
// ===== library: MasterCopy "Copy of Function blocks in 1. FB Bilbiotecas" =====

// folder: 1. FB Bilbiotecas

FUNCTION_BLOCK "FB BITS TO WORD"   // FB1, SCL
{ S7_Optimized_Access := 'TRUE' }
VERSION : 0.1
// Empacota 16 bools numa Word. Contrato consumido por gen-alarm-fc:
//  pinos de entrada SIGNAL_Bit0..SIGNAL_Bit15 e saida BITS_TO_WORD --
//  AlarmFc.RewireWordNetwork procura esses nomes exatos (AlarmFc.cs:313 e :348).
//  Renomear pino aqui quebra o gerador.
   VAR_INPUT
      SIGNAL_Bit0 : Bool;
      SIGNAL_Bit1 : Bool;
      SIGNAL_Bit2 : Bool;
      SIGNAL_Bit3 : Bool;
      SIGNAL_Bit4 : Bool;
      SIGNAL_Bit5 : Bool;
      SIGNAL_Bit6 : Bool;
      SIGNAL_Bit7 : Bool;
      SIGNAL_Bit8 : Bool;
      SIGNAL_Bit9 : Bool;
      SIGNAL_Bit10 : Bool;
      SIGNAL_Bit11 : Bool;
      SIGNAL_Bit12 : Bool;
      SIGNAL_Bit13 : Bool;
      SIGNAL_Bit14 : Bool;
      SIGNAL_Bit15 : Bool;
   END_VAR
   VAR_OUTPUT
      BITS_TO_WORD : Word;
   END_VAR
BEGIN

      // slice access: %X0 e o bit menos significativo da Word
      #BITS_TO_WORD.%X0 := #SIGNAL_Bit0;
      #BITS_TO_WORD.%X1 := #SIGNAL_Bit1;
      #BITS_TO_WORD.%X2 := #SIGNAL_Bit2;
      #BITS_TO_WORD.%X3 := #SIGNAL_Bit3;
      #BITS_TO_WORD.%X4 := #SIGNAL_Bit4;
      #BITS_TO_WORD.%X5 := #SIGNAL_Bit5;
      #BITS_TO_WORD.%X6 := #SIGNAL_Bit6;
      #BITS_TO_WORD.%X7 := #SIGNAL_Bit7;
      #BITS_TO_WORD.%X8 := #SIGNAL_Bit8;
      #BITS_TO_WORD.%X9 := #SIGNAL_Bit9;
      #BITS_TO_WORD.%X10 := #SIGNAL_Bit10;
      #BITS_TO_WORD.%X11 := #SIGNAL_Bit11;
      #BITS_TO_WORD.%X12 := #SIGNAL_Bit12;
      #BITS_TO_WORD.%X13 := #SIGNAL_Bit13;
      #BITS_TO_WORD.%X14 := #SIGNAL_Bit14;
      #BITS_TO_WORD.%X15 := #SIGNAL_Bit15;
END_FUNCTION_BLOCK

FUNCTION_BLOCK "FB BITS TO DOUBLE WORD"   // FB5, SCL
{ S7_Optimized_Access := 'TRUE' }
VERSION : 0.1
   VAR_INPUT
      SIGNAL_Bit0 : Bool;   // Sinal de entrada 1
      SIGNAL_Bit1 : Bool;   // Sinal de entrada 2
      SIGNAL_Bit2 : Bool;   // Sinal de entrada 3
      SIGNAL_Bit3 : Bool;   // Sinal de entrada 4
      SIGNAL_Bit4 : Bool;   // Sinal de entrada 5
      SIGNAL_Bit5 : Bool;   // Sinal de entrada 6
      SIGNAL_Bit6 : Bool;   // Sinal de entrada 7
      SIGNAL_Bit7 : Bool;   // Sinal de entrada 8
      SIGNAL_Bit8 : Bool;   // Sinal de entrada 9
      SIGNAL_Bit9 : Bool;   // Sinal de entrada 10
      SIGNAL_Bit10 : Bool;   // Sinal de entrada 11
      SIGNAL_Bit11 : Bool;   // Sinal de entrada 12
      SIGNAL_Bit12 : Bool;   // Sinal de entrada 13
      SIGNAL_Bit13 : Bool;   // Sinal de entrada 14
      SIGNAL_Bit14 : Bool;   // Sinal de entrada 15
      SIGNAL_Bit15 : Bool;   // Sinal de entrada 16
      SIGNAL_Bit16 : Bool;   // Sinal de entrada 17
      SIGNAL_Bit17 : Bool;   // Sinal de entrada 18
      SIGNAL_Bit18 : Bool;   // Sinal de entrada 19
      SIGNAL_Bit19 : Bool;   // Sinal de entrada 20
      SIGNAL_Bit20 : Bool;   // Sinal de entrada 21
      SIGNAL_Bit21 : Bool;   // Sinal de entrada 22
      SIGNAL_Bit22 : Bool;   // Sinal de entrada 23
      SIGNAL_Bit23 : Bool;   // Sinal de entrada 24
      SIGNAL_Bit24 : Bool;   // Sinal de entrada 25
      SIGNAL_Bit25 : Bool;   // Sinal de entrada 26
      SIGNAL_Bit26 : Bool;   // Sinal de entrada 27
      SIGNAL_Bit27 : Bool;   // Sinal de entrada 28
      SIGNAL_Bit28 : Bool;   // Sinal de entrada 29
      SIGNAL_Bit29 : Bool;   // Sinal de entrada 30
      SIGNAL_Bit30 : Bool;   // Sinal de entrada 31
      SIGNAL_Bit31 : Bool;   // Sinal de entrada 32
   END_VAR
   VAR_OUTPUT
      BITS_TO_DWORD : DWord;   // Word de saída com os sinais montados
   END_VAR
BEGIN
   // Word Alarmes - Montando bits em uma double word

   // Bits recebidos de campo
   #"BITS_TO_DWORD".%X0 := #SIGNAL_Bit0;
   #"BITS_TO_DWORD".%X1 := #SIGNAL_Bit1;
   #"BITS_TO_DWORD".%X2 := #SIGNAL_Bit2;
   #"BITS_TO_DWORD".%X3 := #SIGNAL_Bit3;
   #"BITS_TO_DWORD".%X4 := #SIGNAL_Bit4;
   #"BITS_TO_DWORD".%X5 := #SIGNAL_Bit5;
   #"BITS_TO_DWORD".%X6 := #SIGNAL_Bit6;
   #"BITS_TO_DWORD".%X7 := #SIGNAL_Bit7;
   #"BITS_TO_DWORD".%X8 := #SIGNAL_Bit8;
   #"BITS_TO_DWORD".%X9 := #SIGNAL_Bit9;
   #"BITS_TO_DWORD".%X10 := #SIGNAL_Bit10;
   #"BITS_TO_DWORD".%X11 := #SIGNAL_Bit11;
   #"BITS_TO_DWORD".%X12 := #SIGNAL_Bit12;
   #"BITS_TO_DWORD".%X13 := #SIGNAL_Bit13;
   #"BITS_TO_DWORD".%X14 := #SIGNAL_Bit14;
   #"BITS_TO_DWORD".%X15 := #SIGNAL_Bit15;
   #"BITS_TO_DWORD".%X16 := #SIGNAL_Bit16;
   #"BITS_TO_DWORD".%X17 := #SIGNAL_Bit17;
   #"BITS_TO_DWORD".%X18 := #SIGNAL_Bit18;
   #"BITS_TO_DWORD".%X19 := #SIGNAL_Bit19;
   #"BITS_TO_DWORD".%X20 := #SIGNAL_Bit20;
   #"BITS_TO_DWORD".%X21 := #SIGNAL_Bit21;
   #"BITS_TO_DWORD".%X22 := #SIGNAL_Bit22;
   #"BITS_TO_DWORD".%X23 := #SIGNAL_Bit23;
   #"BITS_TO_DWORD".%X24 := #SIGNAL_Bit24;
   #"BITS_TO_DWORD".%X25 := #SIGNAL_Bit25;
   #"BITS_TO_DWORD".%X26 := #SIGNAL_Bit26;
   #"BITS_TO_DWORD".%X27 := #SIGNAL_Bit27;
   #"BITS_TO_DWORD".%X28 := #SIGNAL_Bit28;
   #"BITS_TO_DWORD".%X29 := #SIGNAL_Bit29;
   #"BITS_TO_DWORD".%X30 := #SIGNAL_Bit30;
   #"BITS_TO_DWORD".%X31 := #SIGNAL_Bit31;
END_FUNCTION_BLOCK

FUNCTION_BLOCK "FB CONTADOR"   // FB7, LAD
TITLE = Function Block MINUTEIRO - Contador de Minutos
{ S7_Optimized_Access := 'TRUE' }
VERSION : 0.1
// Bloco para realizar a contagem de quantos minutos cada motor/bomba passou ligado.
   VAR_INPUT
      INPUT_LIGADO : Bool;   // Entrada do sinal de falha instanciado na Network 1
      INPUT_RESET_MINUTEIRO : Bool;   // Entrada do sinal de reset minuteiro (minutos trabalhadas da bomba)
   END_VAR
   VAR_OUTPUT
      SEGUNDEIRO : UInt;   // Saída do segundeiro (segundos trabalhados da bomba)
      MINUTEIRO : Real;   // Saída do minuteiro (minutos trabalhados da bomba)
      HORIMETRO : Real;   // Saída do horimetro (horas trabalhados da bomba)
   END_VAR
   VAR
      RESET_SEGUNDO : Bool;   // Comando para zerar os minutos acumuladas
      MINUTO : Bool;   // Pulso para contador de minutos
      COUNT_MINUTO : Bool;   // Contador de minutos
      RESET_MINUTO : Bool;   // Reset do contador de minutos
      SEGUNDOS : UInt;   // Segundos armazenados
      TIMER_SEGUNDO : IEC_COUNTER;   // Bloco contador de segundos
   END_VAR
BEGIN

REGION Network 1: Comando para zerar os minutos acumuladas
   // TIMER_SEGUNDO: Bloco contador de segundos
   // TIMER_MINUTO: Bloco contador de minutos
   // INC: Incremento de horas
   // RESET_MINUTEIRO: Comando para zerar os minutos acumulados
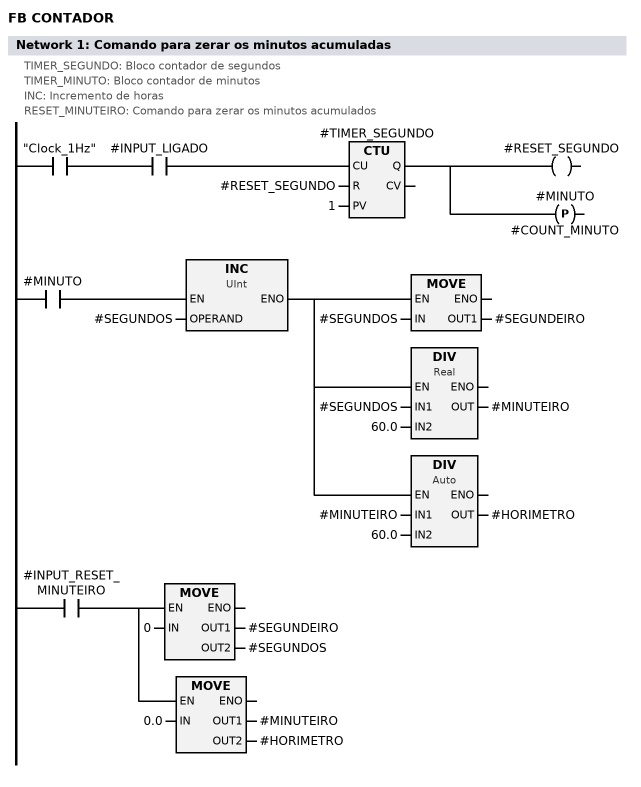
   #TIMER_SEGUNDO.CTU(CU := "Clock_1Hz" AND #INPUT_LIGADO, R := #RESET_SEGUNDO, PV := 1);
   #RESET_SEGUNDO := #TIMER_SEGUNDO.Q;
   #MINUTO := #TIMER_SEGUNDO.Q AND NOT #COUNT_MINUTO;   // rising edge
   #COUNT_MINUTO := #TIMER_SEGUNDO.Q;
   IF #MINUTO THEN
       #SEGUNDOS := #SEGUNDOS + 1;
       #SEGUNDEIRO := #SEGUNDOS;
       #MINUTEIRO := #SEGUNDOS / 60.0;
       #HORIMETRO := #MINUTEIRO / 60.0;
   END_IF;
   IF #INPUT_RESET_MINUTEIRO THEN
       #SEGUNDEIRO := 0;
       #SEGUNDOS := 0;
       #MINUTEIRO := 0.0;
       #HORIMETRO := 0.0;
   END_IF;
END_REGION
END_FUNCTION_BLOCK

FUNCTION_BLOCK "FB TOTALIZADOR"   // FB16, LAD
TITLE = Function Block TOTALIZADOR - Calculando os totalizadores dos macromedidores
{ S7_Optimized_Access := 'TRUE' }
VERSION : 0.1
// Network 1: Recebendo sinal de pulso
// Network 2: Primeira Soma (Incremento a cada 1 pulso)
// Network 3: Segunda Soma (Incremento a cada 1000 pulsos)
// Network 4: Resetando o totalizador
   VAR_INPUT
      ENTRADA_SINAL : Bool;   // Entrada do sinal proveniente do hidrômetro/macromedidor
      RESET_TOT : Bool;   // Input de reset para zerar os blocos de incremento do totalizador
      MULTIPLICADOR : Int;
   END_VAR
   VAR_OUTPUT
      TOT_SAÍDA : UInt;   // Saída real do totalizador (m³)
   END_VAR
   VAR RETAIN
      PULSE1 : Bool;   // Pulso inicial para contar os sinais elétricos da entrada digital
      COUNT_PULSE1 : Bool;   // Contador de Pulsos 1
      PULSE2 : Bool;   // Rampa de subida para assegurar que o sinal da comparação anterior seja identificado como pulso pelo CLP
      COUNT_PULSE2 : Bool;   // Contador de pulsos 2
      SOMA1 : UInt;   // Bloco de incremento a cada pulso recebido na variável PULSE
      SOMA1_TOT_PREV : UInt;   // Variável que recebe a primeira soma
      SOMA2 : UInt;   // Variável que recebe o incremento de 1000 em 1000 e move ao TOT_SAÍDA Output para ser utilizado
   END_VAR
   VAR
      MULT1 : UInt;
   END_VAR
BEGIN

REGION Network 1: Recebendo sinal de pulso
   // ENTRADA_SINAL: Input que recebe o sinal de pulso do equipamento
   // PULSE1: Rampa de subida para assegurar que o sinal recebido seja identificado como pulso pelo CLP
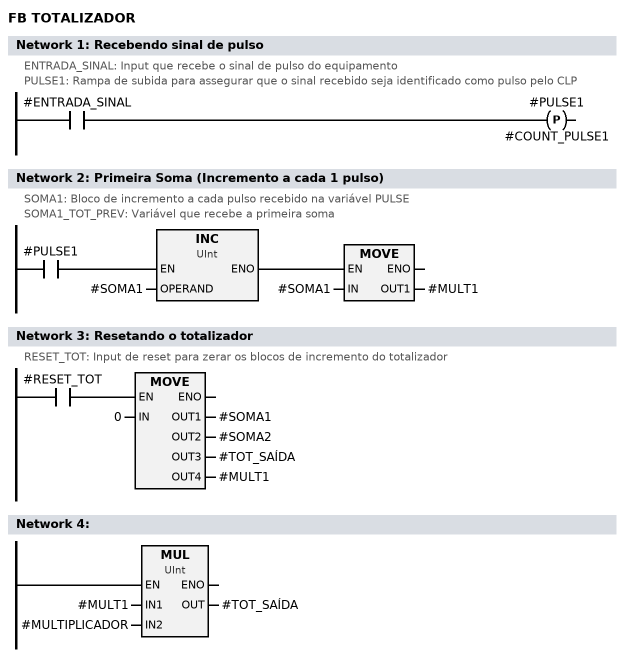
   #PULSE1 := #ENTRADA_SINAL AND NOT #COUNT_PULSE1;   // rising edge
   #COUNT_PULSE1 := #ENTRADA_SINAL;
END_REGION

REGION Network 2: Primeira Soma (Incremento a cada 1 pulso)
   // SOMA1: Bloco de incremento a cada pulso recebido na variável PULSE
   // SOMA1_TOT_PREV: Variável que recebe a primeira soma
   RUNG wire#powerrail
      Contact( #PULSE1 )
      { S7_Templates := "DestType := UInt" } Inc( #SOMA1 )
      Move(in := #SOMA1, out1 => #MULT1)
   END_RUNG
   // the same network as SCL:
   IF #PULSE1 THEN
       #SOMA1 := #SOMA1 + 1;
       #MULT1 := #SOMA1;
   END_IF;
END_REGION

REGION Network 3: Resetando o totalizador
   // RESET_TOT: Input de reset para zerar os blocos de incremento do totalizador
   RUNG wire#powerrail
      Contact( #RESET_TOT )
      Move(in := 0, out1 => #SOMA1, out2 => #SOMA2, out3 => #TOT_SAÍDA, out4 => #MULT1)
   END_RUNG
   // the same network as SCL:
   IF #RESET_TOT THEN
       #SOMA1 := 0;
       #SOMA2 := 0;
       #TOT_SAÍDA := 0;
       #MULT1 := 0;
   END_IF;
END_REGION

REGION Network 4
   RUNG wire#powerrail
      { S7_Templates := "SrcType := UInt" } Mul(in1 := #MULT1, in2 := #MULTIPLICADOR, out => #TOT_SAÍDA)
   END_RUNG
   // the same network as SCL:
   #TOT_SAÍDA := #MULT1 * #MULTIPLICADOR;
END_REGION
END_FUNCTION_BLOCK

FUNCTION_BLOCK "FB_HORÍMETRO"   // FB22, LAD
TITLE = Function Block HORÍMETRO - Contador de Horas
{ S7_Optimized_Access := 'TRUE' }
VERSION : 0.1
// Bloco para realizar a contagem de quantas horas cada motor/bomba passou ligado.
   VAR_INPUT
      INPUT_LIGADO : Bool;   // Entrada do sinal de falha instanciado na Network 1
      INPUT_RESET_HORIMETRO : Bool;   // Entrada do sinal de reset horímetro (horas trabalhadas da bomba)
   END_VAR
   VAR_OUTPUT
      HORIMETRO : UInt;   // Saída do horímetro (horas trabalhadas da bomba)
   END_VAR
   VAR RETAIN
      RESET_SEGUNDO : Bool;   // Comando para zerar as horas acumuladas
      MINUTO : Bool;   // Pulso para contador de minutos
      COUNT_MINUTO : Bool;   // Contador de minutos
      RESET_MINUTO : Bool;   // Reset do contador de minutos
      HORA : Bool;   // Pulso para contador de horas
      COUNT_HORA : Bool;   // Contador de horas
      HORAS : UInt;   // Horas armazenadas para mover ao Horimetro e zerar quando solicitado
      TIMER_SEGUNDO : IEC_COUNTER;   // Bloco contador de segundos
      TIMER_MINUTO : IEC_COUNTER;   // Bloco contador de minutos
   END_VAR
BEGIN

REGION Network 1: Acumulação de horas (Utilizando clock de 1Hz/1s)
   // TIMER_SEGUNDO: Bloco contador de segundos
   // TIMER_MINUTO: Bloco contador de minutos
   // INC: Incremento de horas
   // RESET_HORIMETRO: Comando para zerar as horas acumuladas
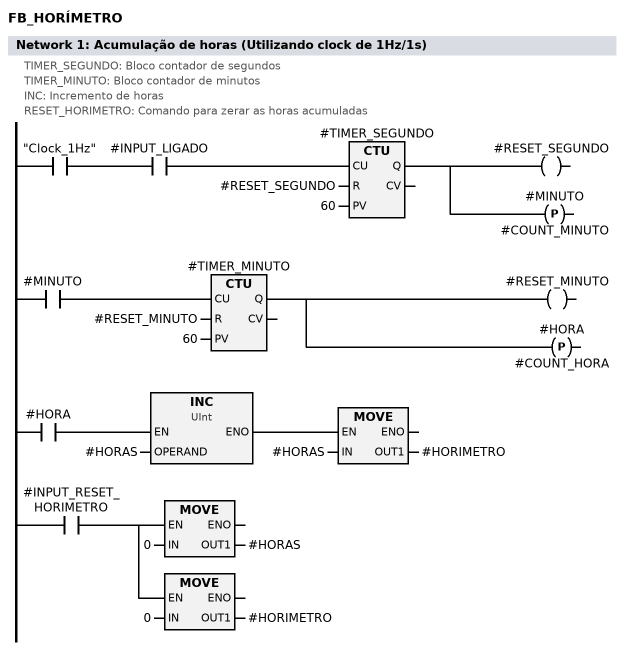
   #TIMER_SEGUNDO.CTU(CU := "Clock_1Hz" AND #INPUT_LIGADO, R := #RESET_SEGUNDO, PV := 60);
   #RESET_SEGUNDO := #TIMER_SEGUNDO.Q;
   #MINUTO := #TIMER_SEGUNDO.Q AND NOT #COUNT_MINUTO;   // rising edge
   #COUNT_MINUTO := #TIMER_SEGUNDO.Q;
   #TIMER_MINUTO.CTU(CU := #MINUTO, R := #RESET_MINUTO, PV := 60);
   #RESET_MINUTO := #TIMER_MINUTO.Q;
   #HORA := #TIMER_MINUTO.Q AND NOT #COUNT_HORA;   // rising edge
   #COUNT_HORA := #TIMER_MINUTO.Q;
   IF #HORA THEN
       #HORAS := #HORAS + 1;
       #HORIMETRO := #HORAS;
   END_IF;
   IF #INPUT_RESET_HORIMETRO THEN
       #HORAS := 0;
       #HORIMETRO := 0;
   END_IF;
END_REGION
END_FUNCTION_BLOCK

// folder: 1. FB Bilbiotecas/1.1 Acionamento

FUNCTION_BLOCK "FB CONDIÇÃO DE PARTIDA"   // FB6, LAD
TITLE = Function Block CONDIÇÃO DE PARTIDA - Intertravamentos para partir o motor/bomba
{ S7_Optimized_Access := 'TRUE' }
VERSION : 0.1
// Network 1: Gerenciamento Status Motor/Bomba
// Network 2: Recebimento dos sinais de entrada (Sinais de campo e comandos)
// Network 3: MODO MANUAL: Conjunto de condições para ligar e desligar
// Network 4: MODO AUTOMÁTICO: Conjunto de condições para ligar e desligar
// Network 5: FALHA: Condicionamento de falha
// Network 6: LIGA BOMBA: Validando intertravamentos para ligar
   VAR_INPUT
      INPUT_LIGADO : Bool;   // 1 = Sinal elétrico de campo indicando bomba ligada
      INPUT_DESLIGADO : Bool;   // 1 = Sinal elétrico de campo indicando bomba desligada
      INPUT_FALHA : Bool;   // 0 = Sinal elétrico de campo indicando bomba em falha
      INPUT_LOCAL_MAN : Bool;   // 1 = Sinal elétrico de campo indicando bomba em local
      INPUT_LOCAL_AUTO : Bool;   // 1 = Sinal elétrico de campo indicando bomba em local automático
      INPUT_REMOTO : Bool;   // 1 = Sinal elétrico de campo indicando bomba em remoto
      INPUT_FALHA_PROFINET : Bool;   // 1 = Indica falta de comunicação PROFINET com o equipamento
      INPUT_HABILITA_LIGA_AUTO : Bool;   // 1 = Sinal para habilitar Liga Bomba em Modo Automático quando todas as condições foram atentidas
      INPUT_CMD_LIGA : Bool;   // Comando enviado da IHM/SCADA para ligar a bomba
      CMD_MANUTEN : Bool;   // Comando enviado da IHM/SCADA para colocar a bomba em Modo de Manutenção
      CMD_MODO_OPERACAO : Bool;   // Comando enviado da IHM/SCADA para colocar a bomba em (0 = Modo Manual, 1 = Modo Automático)
      CMD_RESET_HORIMETRO : Bool;
   END_VAR
   VAR_OUTPUT
      LIGA_BOMBA : Bool;   // Saída acionada para ligar a bomba remotamente
      STATUS_MOTOR : Byte;   // 0 = DESLIGADO; 1 = LIGADO; 2 = FALHA; 3 = MANUTENÇÃO; 4 = SEM COMUNICAÇÃO MODBUS
      OUTPUT_REMOTO_AUTO : Bool;   // Saída para indicar bomba em Remoto Automático
      OUTPUT_MODO_OPER : Byte;
      STS_HORIMETRO : UInt;
      RESET_CMD_LIGA : Bool;
      STS_INTERTRAVAMENTO_AUTOMATICO : Bool;
   END_VAR
   VAR
      LOCAL_MAN : Bool;   // Saída para indicar bomba em Local Manual
      REMOTO_MAN : Bool;   // Saída para indicar bomba em Remoto Manual
      MANUTEN : Bool;   // Variável local para Indicar bomba em Modo Manutenção
      REMOTO : Bool;   // Variável local para indicar bomba em Modo Remoto
      FALHA : Bool;   // Variável local para indicar bomba em Falha
      LOCAL_AUTO : Bool;   // Variável local para indicar bomba em Modo Local Automático
      LIGA_REM_MAN : Bool;   // Variável local para Acionamento Remoto Manual
      LIGA_REM_AUTO : Bool;   // Variável local para Acionamento Remoto Automático
      "FB MODOS DE OPERAÇÃO_Instance" : "FB MODOS DE OPERAÇÃO";
      FB_HORÍMETRO_Instance : "FB_HORÍMETRO";
   END_VAR
   VAR_TEMP   // added for the SCL form of the ladder/FBD networks
      _w1 : Bool;
   END_VAR
BEGIN

REGION Network 1: Recebimento dos sinais de entrada (Sinais de campo e comandos)
   // INPUT_ABERTA = Entrada de sinal de Bomba Ligada
   // INPUT_FECHADA = Entrada de sinal de Bomba Desligada
   // INPUT_FALHA = Entrada de sinal de Bomba em Falha
   // INPUT_FALHA_PROFINET = Sem comunicação Profinet
   // STATUS_MOTOR: 0 = DESLIGADO; 1 = LIGADO; 2 = FALHA; 3 = MANUTENÇÃO; 4 = SEM COMUNICAÇÃO MODBUS
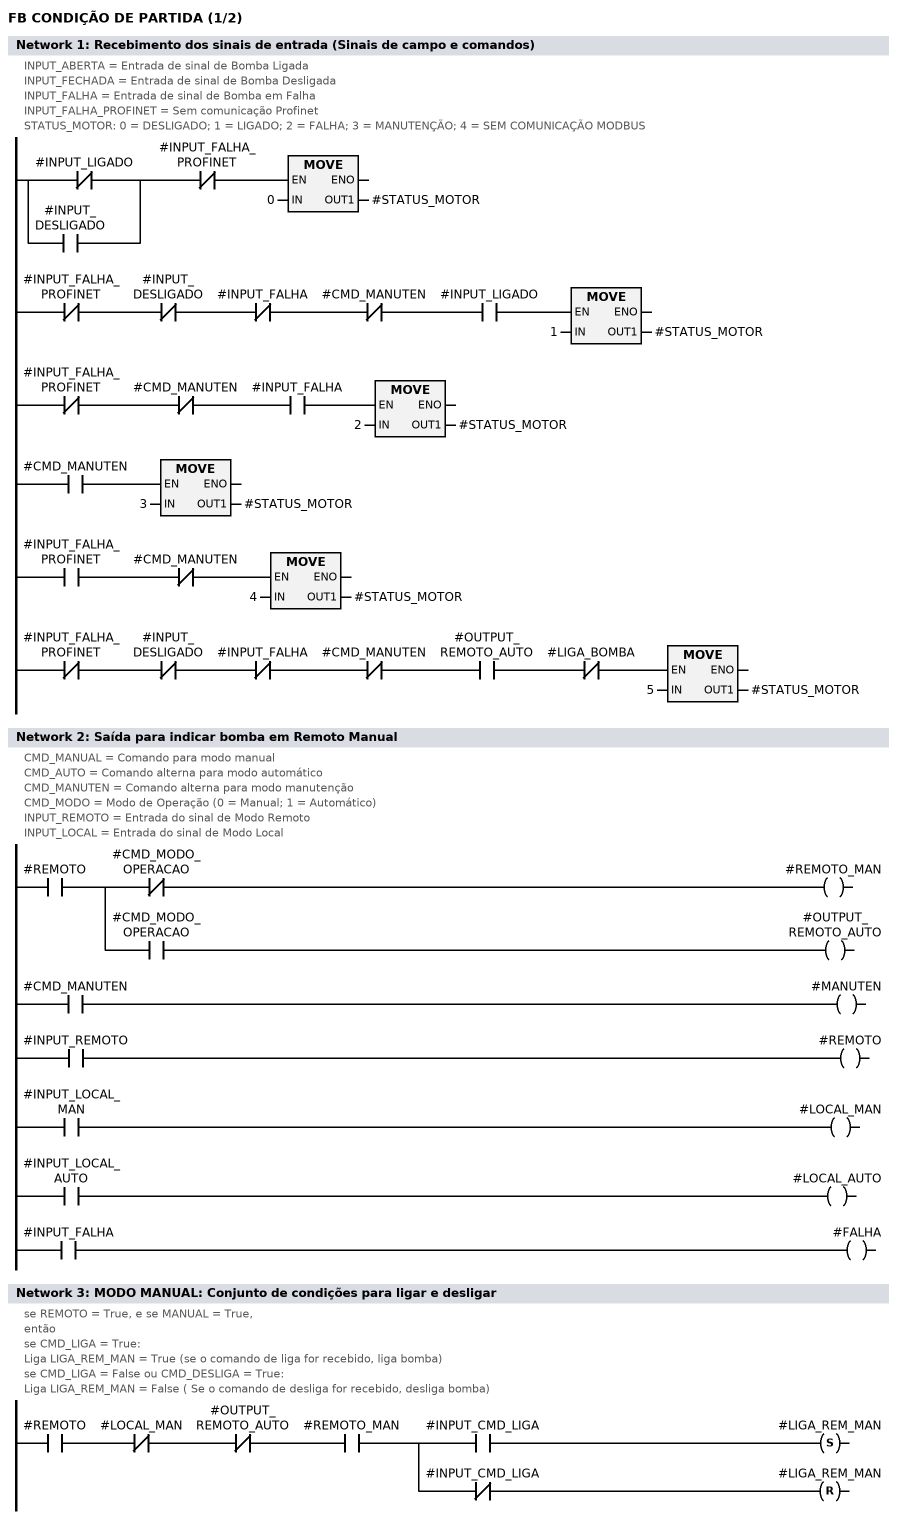
   RUNG wire#powerrail
      I_Contact( #INPUT_LIGADO )
      wire#w1
      I_Contact( #INPUT_FALHA_PROFINET )
      Move(in := 0, out1 => #STATUS_MOTOR)
   END_RUNG
   RUNG wire#powerrail
      Contact( #INPUT_DESLIGADO )
   END_RUNG wire#w1
   RUNG wire#powerrail
      I_Contact( #INPUT_FALHA_PROFINET )
      I_Contact( #INPUT_DESLIGADO )
      I_Contact( #INPUT_FALHA )
      I_Contact( #CMD_MANUTEN )
      Contact( #INPUT_LIGADO )
      Move(in := 1, out1 => #STATUS_MOTOR)
   END_RUNG
   RUNG wire#powerrail
      I_Contact( #INPUT_FALHA_PROFINET )
      I_Contact( #CMD_MANUTEN )
      Contact( #INPUT_FALHA )
      Move(in := 2, out1 => #STATUS_MOTOR)
   END_RUNG
   RUNG wire#powerrail
      Contact( #CMD_MANUTEN )
      Move(in := 3, out1 => #STATUS_MOTOR)
   END_RUNG
   RUNG wire#powerrail
      Contact( #INPUT_FALHA_PROFINET )
      I_Contact( #CMD_MANUTEN )
      Move(in := 4, out1 => #STATUS_MOTOR)
   END_RUNG
   RUNG wire#powerrail
      I_Contact( #INPUT_FALHA_PROFINET )
      I_Contact( #INPUT_DESLIGADO )
      I_Contact( #INPUT_FALHA )
      I_Contact( #CMD_MANUTEN )
      Contact( #OUTPUT_REMOTO_AUTO )
      I_Contact( #LIGA_BOMBA )
      Move(in := 5, out1 => #STATUS_MOTOR)
   END_RUNG
   // the same network as SCL:
   IF (NOT #INPUT_LIGADO OR #INPUT_DESLIGADO) AND NOT #INPUT_FALHA_PROFINET THEN #STATUS_MOTOR := 0; END_IF;
   IF NOT #INPUT_FALHA_PROFINET AND NOT #INPUT_DESLIGADO AND NOT #INPUT_FALHA AND NOT #CMD_MANUTEN AND #INPUT_LIGADO THEN
       #STATUS_MOTOR := 1;
   END_IF;
   IF NOT #INPUT_FALHA_PROFINET AND NOT #CMD_MANUTEN AND #INPUT_FALHA THEN #STATUS_MOTOR := 2; END_IF;
   IF #CMD_MANUTEN THEN #STATUS_MOTOR := 3; END_IF;
   IF #INPUT_FALHA_PROFINET AND NOT #CMD_MANUTEN THEN #STATUS_MOTOR := 4; END_IF;
   IF NOT #INPUT_FALHA_PROFINET AND NOT #INPUT_DESLIGADO AND NOT #INPUT_FALHA AND NOT #CMD_MANUTEN AND #OUTPUT_REMOTO_AUTO AND NOT #LIGA_BOMBA THEN
       #STATUS_MOTOR := 5;
   END_IF;
END_REGION

REGION Network 2: Saída para indicar bomba em Remoto Manual
   // CMD_MANUAL = Comando para modo manual
   // CMD_AUTO = Comando alterna para modo automático
   // CMD_MANUTEN = Comando alterna para modo manutenção
   // CMD_MODO = Modo de Operação (0 = Manual; 1 = Automático)
   // INPUT_REMOTO = Entrada do sinal de Modo Remoto
   // INPUT_LOCAL = Entrada do sinal de Modo Local
   RUNG wire#powerrail
      Contact( #REMOTO )
      wire#w1
      I_Contact( #CMD_MODO_OPERACAO )
      Coil( #REMOTO_MAN )
   END_RUNG
   RUNG wire#w1
      Contact( #CMD_MODO_OPERACAO )
      Coil( #OUTPUT_REMOTO_AUTO )
   END_RUNG
   RUNG wire#powerrail
      Contact( #CMD_MANUTEN )
      Coil( #MANUTEN )
   END_RUNG
   RUNG wire#powerrail
      Contact( #INPUT_REMOTO )
      Coil( #REMOTO )
   END_RUNG
   RUNG wire#powerrail
      Contact( #INPUT_LOCAL_MAN )
      Coil( #LOCAL_MAN )
   END_RUNG
   RUNG wire#powerrail
      Contact( #INPUT_LOCAL_AUTO )
      Coil( #LOCAL_AUTO )
   END_RUNG
   RUNG wire#powerrail
      Contact( #INPUT_FALHA )
      Coil( #FALHA )
   END_RUNG
   // the same network as SCL:
   #REMOTO_MAN := #REMOTO AND NOT #CMD_MODO_OPERACAO;
   #OUTPUT_REMOTO_AUTO := #REMOTO AND #CMD_MODO_OPERACAO;
   #MANUTEN := #CMD_MANUTEN;
   #REMOTO := #INPUT_REMOTO;
   #LOCAL_MAN := #INPUT_LOCAL_MAN;
   #LOCAL_AUTO := #INPUT_LOCAL_AUTO;
   #FALHA := #INPUT_FALHA;
END_REGION

REGION Network 3: MODO MANUAL: Conjunto de condições para ligar e desligar
   // se REMOTO = True, e se MANUAL = True,
   // 
   // então
   // se CMD_LIGA = True: 
   // Liga LIGA_REM_MAN = True (se o comando de liga for recebido, liga bomba)
   // 
   // se CMD_LIGA = False ou CMD_DESLIGA = True:
   // Liga LIGA_REM_MAN = False ( Se o comando de desliga for recebido, desliga bomba)
   RUNG wire#powerrail
      Contact( #REMOTO )
      I_Contact( #LOCAL_MAN )
      I_Contact( #OUTPUT_REMOTO_AUTO )
      Contact( #REMOTO_MAN )
      wire#w1
      Contact( #INPUT_CMD_LIGA )
      S_Coil( #LIGA_REM_MAN )
   END_RUNG
   RUNG wire#w1
      I_Contact( #INPUT_CMD_LIGA )
      R_Coil( #LIGA_REM_MAN )
   END_RUNG
   // the same network as SCL:
   #_w1 := #REMOTO AND NOT #LOCAL_MAN AND NOT #OUTPUT_REMOTO_AUTO AND #REMOTO_MAN;
   IF #_w1 AND #INPUT_CMD_LIGA THEN #LIGA_REM_MAN := TRUE; END_IF;
   IF #_w1 AND NOT #INPUT_CMD_LIGA THEN #LIGA_REM_MAN := FALSE; END_IF;
END_REGION

REGION Network 4: Variável local para Acionamento Remoto Auto
   // se REMOTO = True, e se AUTO = True:
   // 
   // então
   // se LIGA_REM_AUTO = True:
   // e se PARAMETRO < PARAMETRO_LIGA;
   // então LIGA_REM_AUTO = True (se a leitura for menor que o cadastro para ligar, liga em remoto automático)
   // 
   // se LIGA_REM_AUTO = False:
   // e se PARAMETRO >= PARAMETRO_DESLIGA:
   // então Desliga REMOTO AUTOMÁTICO (se a leitura for maior ou igual ao cadastro para desligar, desliga em remoto automático)
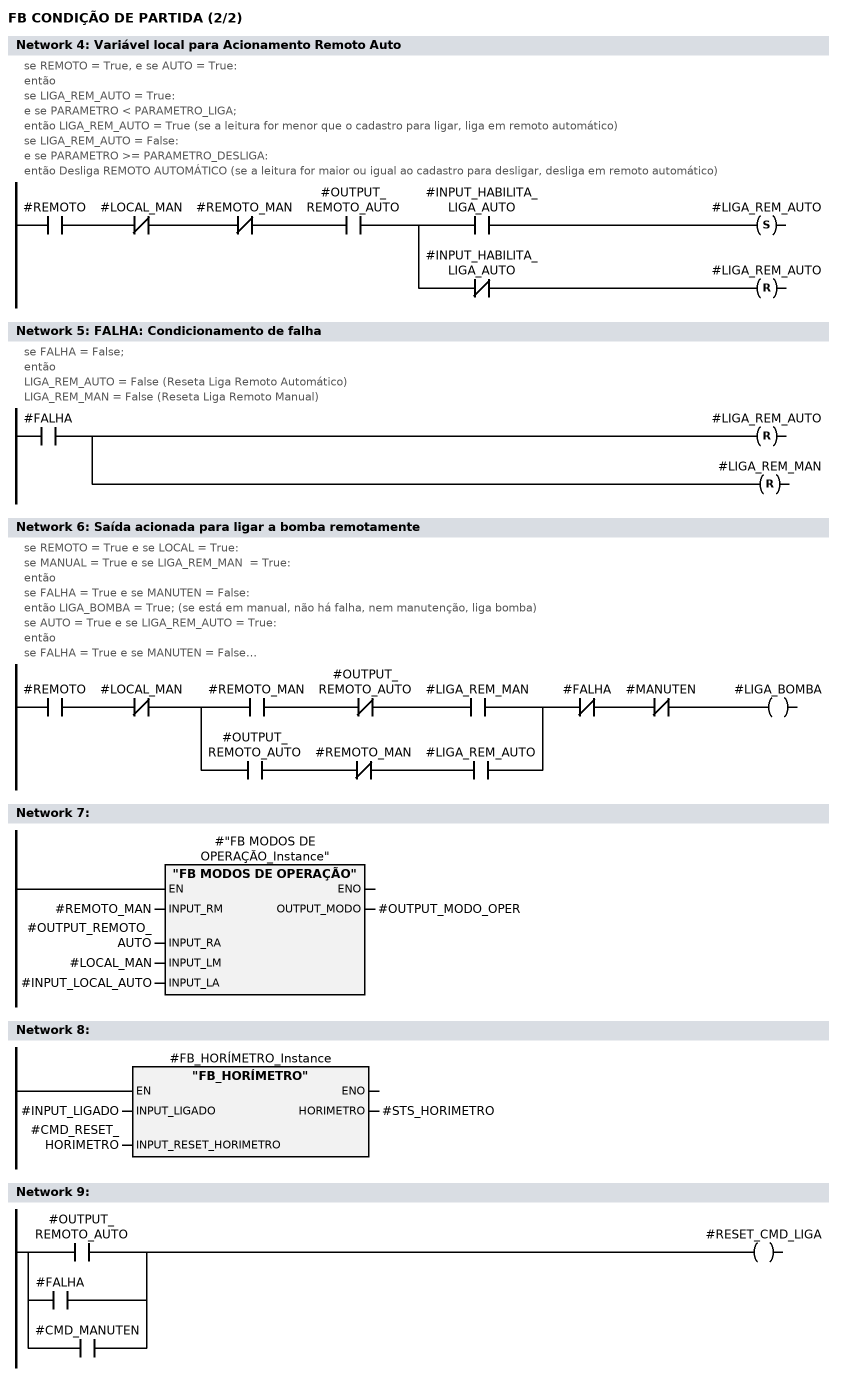
   RUNG wire#powerrail
      Contact( #REMOTO )
      I_Contact( #LOCAL_MAN )
      I_Contact( #REMOTO_MAN )
      Contact( #OUTPUT_REMOTO_AUTO )
      wire#w1
      Contact( #INPUT_HABILITA_LIGA_AUTO )
      S_Coil( #LIGA_REM_AUTO )
   END_RUNG
   RUNG wire#w1
      I_Contact( #INPUT_HABILITA_LIGA_AUTO )
      R_Coil( #LIGA_REM_AUTO )
   END_RUNG
   // the same network as SCL:
   #_w1 := #REMOTO AND NOT #LOCAL_MAN AND NOT #REMOTO_MAN AND #OUTPUT_REMOTO_AUTO;
   IF #_w1 AND #INPUT_HABILITA_LIGA_AUTO THEN #LIGA_REM_AUTO := TRUE; END_IF;
   IF #_w1 AND NOT #INPUT_HABILITA_LIGA_AUTO THEN #LIGA_REM_AUTO := FALSE; END_IF;
END_REGION

REGION Network 5: FALHA: Condicionamento de falha
   // se FALHA = False;
   // 
   // então
   // LIGA_REM_AUTO = False (Reseta Liga Remoto Automático)
   // LIGA_REM_MAN = False (Reseta Liga Remoto Manual)
   RUNG wire#powerrail
      Contact( #FALHA )
      wire#w1
      R_Coil( #LIGA_REM_AUTO )
   END_RUNG
   RUNG wire#w1
      R_Coil( #LIGA_REM_MAN )
   END_RUNG
   // the same network as SCL:
   IF #FALHA THEN
       #LIGA_REM_AUTO := FALSE;
       #LIGA_REM_MAN := FALSE;
   END_IF;
END_REGION

REGION Network 6: Saída acionada para ligar a bomba remotamente
   // se REMOTO = True e se LOCAL = True:
   // 
   // se MANUAL = True e se LIGA_REM_MAN  = True:
   // então
   // se FALHA = True e se MANUTEN = False:
   // então LIGA_BOMBA = True; (se está em manual, não há falha, nem manutenção, liga bomba)
   // 
   // se AUTO = True e se LIGA_REM_AUTO = True:
   // então
   // se FALHA = True e se MANUTEN = False:
   // então LIGA_BOMBA = True; (se está em automático, não há falha, nem manutenção, liga bomba)
   RUNG wire#powerrail
      Contact( #REMOTO )
      I_Contact( #LOCAL_MAN )
      wire#w1
      Contact( #REMOTO_MAN )
      I_Contact( #OUTPUT_REMOTO_AUTO )
      Contact( #LIGA_REM_MAN )
      wire#w2
      I_Contact( #FALHA )
      I_Contact( #MANUTEN )
      Coil( #LIGA_BOMBA )
   END_RUNG
   RUNG wire#w1
      Contact( #OUTPUT_REMOTO_AUTO )
      I_Contact( #REMOTO_MAN )
      Contact( #LIGA_REM_AUTO )
   END_RUNG wire#w2
   // the same network as SCL:
   #LIGA_BOMBA := #REMOTO AND NOT #LOCAL_MAN AND ((#REMOTO_MAN AND NOT #OUTPUT_REMOTO_AUTO AND #LIGA_REM_MAN) OR (#OUTPUT_REMOTO_AUTO AND NOT #REMOTO_MAN AND #LIGA_REM_AUTO)) AND NOT #FALHA AND NOT #MANUTEN;
END_REGION

REGION Network 7
   RUNG wire#powerrail
      #"FB MODOS DE OPERAÇÃO_Instance"(INPUT_RM := #REMOTO_MAN, INPUT_RA := #OUTPUT_REMOTO_AUTO, INPUT_LM := #LOCAL_MAN, INPUT_LA := #INPUT_LOCAL_AUTO, OUTPUT_MODO => #OUTPUT_MODO_OPER)
   END_RUNG
   // the same network as SCL:
   #"FB MODOS DE OPERAÇÃO_Instance"(INPUT_RM := #REMOTO_MAN,   // "FB MODOS DE OPERAÇÃO"
                           INPUT_RA := #OUTPUT_REMOTO_AUTO,
                           INPUT_LM := #LOCAL_MAN,
                           INPUT_LA := #INPUT_LOCAL_AUTO,
                           OUTPUT_MODO => #OUTPUT_MODO_OPER);
END_REGION

REGION Network 8
   RUNG wire#powerrail
      #FB_HORÍMETRO_Instance(INPUT_LIGADO := #INPUT_LIGADO, INPUT_RESET_HORIMETRO := #CMD_RESET_HORIMETRO, HORIMETRO => #STS_HORIMETRO)
   END_RUNG
   // the same network as SCL:
   #FB_HORÍMETRO_Instance(INPUT_LIGADO := #INPUT_LIGADO,   // "FB_HORÍMETRO"
                          INPUT_RESET_HORIMETRO := #CMD_RESET_HORIMETRO,
                          HORIMETRO => #STS_HORIMETRO);
END_REGION

REGION Network 9
   RUNG wire#powerrail
      Contact( #OUTPUT_REMOTO_AUTO )
      wire#w1
      Coil( #RESET_CMD_LIGA )
   END_RUNG
   RUNG wire#powerrail
      Contact( #FALHA )
   END_RUNG wire#w1
   RUNG wire#powerrail
      Contact( #CMD_MANUTEN )
   END_RUNG wire#w1
   // the same network as SCL:
   #RESET_CMD_LIGA := #OUTPUT_REMOTO_AUTO OR #FALHA OR #CMD_MANUTEN;
END_REGION
END_FUNCTION_BLOCK

FUNCTION_BLOCK "FB_LIGA/DESLIGA MODO AUTO"   // FB8, LAD
TITLE = Function Block LIGA/DESLIGA MODO AUTO
{ S7_Optimized_Access := 'TRUE' }
VERSION : 0.1
// Bloco para alternância dinâmica do tempo para ligar e desligar bomba.
// Network 1: Atribuição do sinal de liga
// Network 2: Function Block CONTADOR: Contador de tempo para bomba ligada
// Network 3: Comparativo de bomba ligada com tempo cadastrado para ficar ligada
// Network 4: Function Block CONTADOR: Contador de tempo para bomba desligada
// Network 5: Comparativo de bomba desligada com tempo cadastrado para ficar desligada
// Network 6: Transferindo sinal de bomba ligada/desligada para fora do bloco
   VAR_INPUT
      REMOTO_AUTO : Bool;   // Modo Remoto Automático
      CAD_TEMPO_LIGADA : Real;   // Cadastro tempo para bomba ficar ligada
      CAD_TEMPO_DESLIGADA : Real;   // Cadastro tempo para bomba ficar desligada
      TEMPO_ALTERNANCIA : Bool;   // Controle de alternancia entre bombas
   END_VAR
   VAR_OUTPUT
      HABILITA_LIGA_AUTO : Bool;   // Habilita Liga em Modo Automático
   END_VAR
   VAR_IN_OUT
      TEMPO_LIGADA_AUTO_SEG : Real;   // Tempo de bomba ligada em Modo Automático (segundos)
      TEMPO_LIGADA_AUTO_MIN : Real;   // Tempo de bomba ligada em Modo Automático (minutos)
      TEMPO_LIGADA_AUTO_HOR : Real;   // Tempo de bomba ligada em Modo Automático (horas)
      TEMPO_DESLIGADA_AUTO_SEG : Real;   // Tempo de bomba desligada em Modo Automático (segundos)
      TEMPO_DESLIGADA_AUTO_MIN : Real;   // Tempo de bomba desligada em Modo Automático (minutos)
      TEMPO_DESLIGADA_AUTO_HOR : Real;   // Tempo de bomba desligada em Modo Automático (horas)
   END_VAR
   VAR
      DESLIGA_AUTO : Bool;   // Desliga bomba em Modo Automático
      LIGA_AUTO : Bool;   // Liga bomba em Modo Automático
      MINUTEIRO_LIGADA : "FB CONTADOR";
      MINUTEIRO_DESLIGADA : "FB CONTADOR";
      TEMPO_LIGADA_AUTO_HORA : Bool;   // Tempo de bomba desligada em Modo Automático (em horas)
   END_VAR
BEGIN

REGION Network 1: Atribuição do sinal de liga
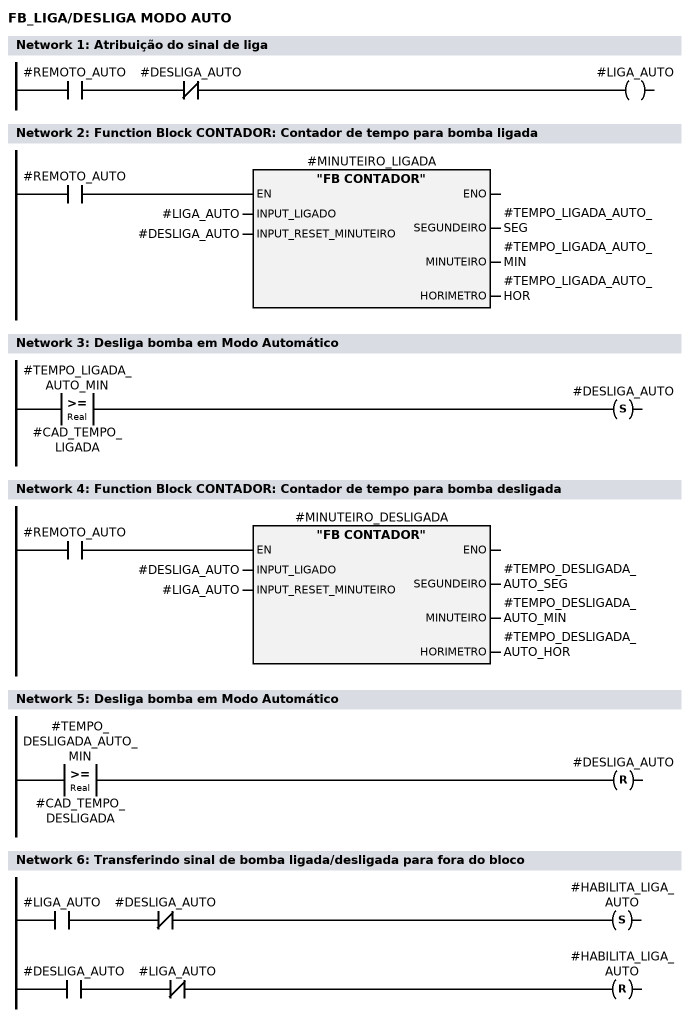
   RUNG wire#powerrail
      Contact( #REMOTO_AUTO )
      I_Contact( #DESLIGA_AUTO )
      Coil( #LIGA_AUTO )
   END_RUNG
   // the same network as SCL:
   #LIGA_AUTO := #REMOTO_AUTO AND NOT #DESLIGA_AUTO;
END_REGION

REGION Network 2: Function Block CONTADOR: Contador de tempo para bomba ligada
   RUNG wire#powerrail
      Contact( #REMOTO_AUTO )
      #MINUTEIRO_LIGADA(INPUT_LIGADO := #LIGA_AUTO, INPUT_RESET_MINUTEIRO := #DESLIGA_AUTO, SEGUNDEIRO => #TEMPO_LIGADA_AUTO_SEG, MINUTEIRO => #TEMPO_LIGADA_AUTO_MIN, HORIMETRO => #TEMPO_LIGADA_AUTO_HOR)
   END_RUNG
   // the same network as SCL:
   IF #REMOTO_AUTO THEN
       #MINUTEIRO_LIGADA(INPUT_LIGADO := #LIGA_AUTO,   // "FB CONTADOR"
                         INPUT_RESET_MINUTEIRO := #DESLIGA_AUTO,
                         SEGUNDEIRO => #TEMPO_LIGADA_AUTO_SEG,
                         MINUTEIRO => #TEMPO_LIGADA_AUTO_MIN,
                         HORIMETRO => #TEMPO_LIGADA_AUTO_HOR);
   END_IF;
END_REGION

REGION Network 3: Desliga bomba em Modo Automático
   RUNG wire#powerrail
      { S7_Templates := "SrcType := Real" } GE_Contact(in1 := #TEMPO_LIGADA_AUTO_MIN, in2 := #CAD_TEMPO_LIGADA)
      S_Coil( #DESLIGA_AUTO )
   END_RUNG
   // the same network as SCL:
   IF #TEMPO_LIGADA_AUTO_MIN >= #CAD_TEMPO_LIGADA THEN #DESLIGA_AUTO := TRUE; END_IF;
END_REGION

REGION Network 4: Function Block CONTADOR: Contador de tempo para bomba desligada
   RUNG wire#powerrail
      Contact( #REMOTO_AUTO )
      #MINUTEIRO_DESLIGADA(INPUT_LIGADO := #DESLIGA_AUTO, INPUT_RESET_MINUTEIRO := #LIGA_AUTO, SEGUNDEIRO => #TEMPO_DESLIGADA_AUTO_SEG, MINUTEIRO => #TEMPO_DESLIGADA_AUTO_MIN, HORIMETRO => #TEMPO_DESLIGADA_AUTO_HOR)
   END_RUNG
   // the same network as SCL:
   IF #REMOTO_AUTO THEN
       #MINUTEIRO_DESLIGADA(INPUT_LIGADO := #DESLIGA_AUTO,   // "FB CONTADOR"
                            INPUT_RESET_MINUTEIRO := #LIGA_AUTO,
                            SEGUNDEIRO => #TEMPO_DESLIGADA_AUTO_SEG,
                            MINUTEIRO => #TEMPO_DESLIGADA_AUTO_MIN,
                            HORIMETRO => #TEMPO_DESLIGADA_AUTO_HOR);
   END_IF;
END_REGION

REGION Network 5: Desliga bomba em Modo Automático
   RUNG wire#powerrail
      { S7_Templates := "SrcType := Real" } GE_Contact(in1 := #TEMPO_DESLIGADA_AUTO_MIN, in2 := #CAD_TEMPO_DESLIGADA)
      R_Coil( #DESLIGA_AUTO )
   END_RUNG
   // the same network as SCL:
   IF #TEMPO_DESLIGADA_AUTO_MIN >= #CAD_TEMPO_DESLIGADA THEN #DESLIGA_AUTO := FALSE; END_IF;
END_REGION

REGION Network 6: Transferindo sinal de bomba ligada/desligada para fora do bloco
   RUNG wire#powerrail
      Contact( #LIGA_AUTO )
      I_Contact( #DESLIGA_AUTO )
      S_Coil( #HABILITA_LIGA_AUTO )
   END_RUNG
   RUNG wire#powerrail
      Contact( #DESLIGA_AUTO )
      I_Contact( #LIGA_AUTO )
      R_Coil( #HABILITA_LIGA_AUTO )
   END_RUNG
   // the same network as SCL:
   IF #LIGA_AUTO AND NOT #DESLIGA_AUTO THEN #HABILITA_LIGA_AUTO := TRUE; END_IF;
   IF #DESLIGA_AUTO AND NOT #LIGA_AUTO THEN #HABILITA_LIGA_AUTO := FALSE; END_IF;
END_REGION
END_FUNCTION_BLOCK

FUNCTION_BLOCK "FB MODOS DE OPERAÇÃO"   // FB10, LAD
TITLE = Function Block MODOS DE OPERAÇÃO
{ S7_Optimized_Access := 'TRUE' }
VERSION : 0.1
// Movendo os valores booleados para uma variável do tipo int
   VAR_INPUT
      INPUT_RM : Bool;   // Entrada de sinal alto para indicar modo Remoto Manual
      INPUT_RA : Bool;   // Entrada de sinal alto para indicar modo Remoto Automático
      INPUT_LM : Bool;   // Entrada de sinal alto para indicar modo Local Manual
      INPUT_LA : Bool;   // Entrada de sinal alto para indicar modo Local Automático
   END_VAR
   VAR_OUTPUT
      OUTPUT_MODO : Int;   // Saída do Modo de Operação
   END_VAR
BEGIN

REGION Network 1: Estrutura de Operação
   // Se Remoto Manual = TRUE, OPERACAO_MOTOR = 1 
   // Se Remoto Automático = TRUE, OPERACAO_MOTOR = 2
   // Se Local Automático = TRUE, OPERACAO_MOTOR = 3
   // Se Local Manual = TRUE, OPERACAO_MOTOR = 4
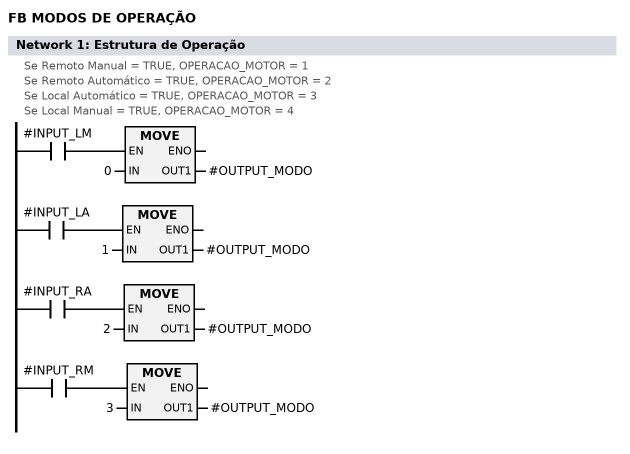
   RUNG wire#powerrail
      Contact( #INPUT_LM )
      Move(in := 0, out1 => #OUTPUT_MODO)
   END_RUNG
   RUNG wire#powerrail
      Contact( #INPUT_LA )
      Move(in := 1, out1 => #OUTPUT_MODO)
   END_RUNG
   RUNG wire#powerrail
      Contact( #INPUT_RA )
      Move(in := 2, out1 => #OUTPUT_MODO)
   END_RUNG
   RUNG wire#powerrail
      Contact( #INPUT_RM )
      Move(in := 3, out1 => #OUTPUT_MODO)
   END_RUNG
   // the same network as SCL:
   IF #INPUT_LM THEN #OUTPUT_MODO := 0; END_IF;
   IF #INPUT_LA THEN #OUTPUT_MODO := 1; END_IF;
   IF #INPUT_RA THEN #OUTPUT_MODO := 2; END_IF;
   IF #INPUT_RM THEN #OUTPUT_MODO := 3; END_IF;
END_REGION
END_FUNCTION_BLOCK

FUNCTION_BLOCK "FB_PARTIDA_INVERSOR"   // FB11, LAD
TITLE = Function Block PARTIDA INVERSOR
{ S7_Optimized_Access := 'TRUE' }
VERSION : 0.1
// Bloco para configurar os sinais de pulso (liga e desliga) em conjunto com 2 relés
   VAR_INPUT
      IN_LIGA_BOMBA : Bool;   // Entrada do comando para ligar a bomba
      IN_SUCÇÃO_OK : Bool;   // 0 = Sucção OK, permite ligar a bomba
      IN_OBSTRUÇÃO : Bool;   // 0 = Obstrução na pista
      IN_SOBRETORQUE : Bool;   // 0 = Sobretorque do motor/bomba
      IN_FALHA : Bool;   // 1 = Bomba em falha, comando desliga é pulsado
      IN_LIGADO : Bool;   // 1 = Bomba Ligada
      IN_HABILITA_CMB : Bool;   // Habilita bomba (Principal / Reserva)
      IN_LIGA_BOMBA_AUTO : Bool;
   END_VAR
   VAR_OUTPUT
      OUT_LIGA : Bool;   // Saída digital para ligar o Inversor
      OUT_DESLIGA : Bool;   // Saída digital para desligar o Inversor
   END_VAR
   VAR
      TEMP_LIGA : IEC_TIMER;   // Temporizador para simular o pulso de liga (0.5s)
      TEMP_DESLIGA : IEC_TIMER;   // Temporizador para simular o pulso de desliga (0.5s)
      DESLIGA_BOMBA : Bool;   // Memória auxiliar para desligar o Inversor
      OUT_TEST : Bool;
   END_VAR
BEGIN

REGION Network 1: Saída digital para ligar o Inversor
   // Condições para ligar:
   // IN_LIGA_BOMBA = 1, Sinal de liga recebido do bloco CONDIÇÃO DE PARTIDA
   // IN_SUCÇÃO = 1, Significa que a bomba está com sucção OK
   // IN_OBSTRUÇÃO = 0, Significa que não há obstrução na pista
   // IN_SOBRETORQUE = 0, Significa que não há alarme de sobretorque do motor/bomba
   // OUT_DESLIGA = 1, Para ligar, é necessário que a entrada digital de desliga no inversor (STOP) esteja com sinal alto, 
   // aguardando que o mesmo seja cortado com um pulso para desligar.
   // - Para desligar é necessário que o motor/bomba esteja enviando sinal de ligado.
   // 
   // Pulso para ligar: Configurado com um tempo de 0.5S
   // Pulso para desligar: Configurado com um tempo de 0.5S
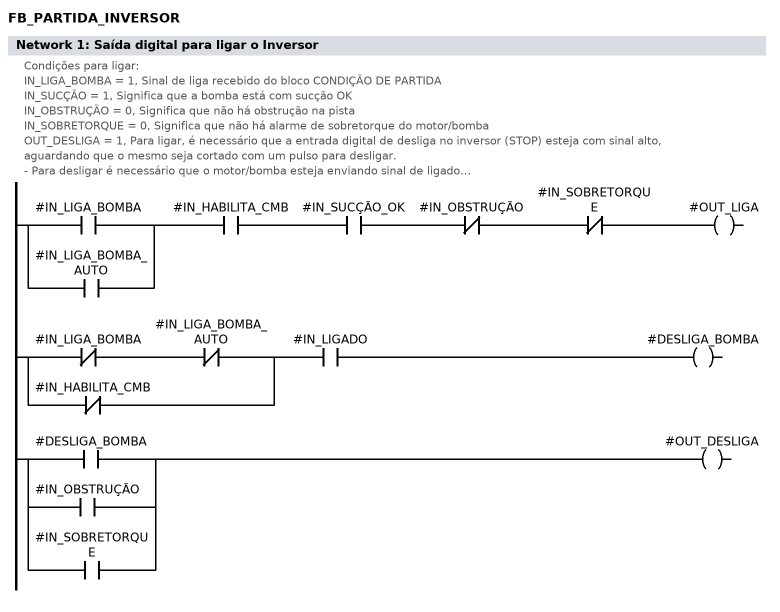
   RUNG wire#powerrail
      Contact( #IN_LIGA_BOMBA )
      wire#w1
      Contact( #IN_HABILITA_CMB )
      Contact( #IN_SUCÇÃO_OK )
      I_Contact( #IN_OBSTRUÇÃO )
      I_Contact( #IN_SOBRETORQUE )
      Coil( #OUT_LIGA )
   END_RUNG
   RUNG wire#powerrail
      Contact( #IN_LIGA_BOMBA_AUTO )
   END_RUNG wire#w1
   RUNG wire#powerrail
      I_Contact( #IN_LIGA_BOMBA )
      I_Contact( #IN_LIGA_BOMBA_AUTO )
      wire#w2
      Contact( #IN_LIGADO )
      Coil( #DESLIGA_BOMBA )
   END_RUNG
   RUNG wire#powerrail
      I_Contact( #IN_HABILITA_CMB )
   END_RUNG wire#w2
   RUNG wire#powerrail
      Contact( #DESLIGA_BOMBA )
      wire#w3
      Coil( #OUT_DESLIGA )
   END_RUNG
   RUNG wire#powerrail
      Contact( #IN_OBSTRUÇÃO )
   END_RUNG wire#w3
   RUNG wire#powerrail
      Contact( #IN_SOBRETORQUE )
   END_RUNG wire#w3
   // the same network as SCL:
   #OUT_LIGA := (#IN_LIGA_BOMBA OR #IN_LIGA_BOMBA_AUTO) AND #IN_HABILITA_CMB AND #IN_SUCÇÃO_OK AND NOT #IN_OBSTRUÇÃO AND NOT #IN_SOBRETORQUE;
   #DESLIGA_BOMBA := ((NOT #IN_LIGA_BOMBA AND NOT #IN_LIGA_BOMBA_AUTO) OR NOT #IN_HABILITA_CMB) AND #IN_LIGADO;
   #OUT_DESLIGA := #DESLIGA_BOMBA OR #IN_OBSTRUÇÃO OR #IN_SOBRETORQUE;
END_REGION
END_FUNCTION_BLOCK

FUNCTION_BLOCK "FB SUCÇÃO OK"   // FB15, LAD
TITLE = Function Block FB SUCÇÃO OK
{ S7_Optimized_Access := 'TRUE' }
VERSION : 0.1
   VAR_INPUT
      REFERENCIA : Real;   // Referência analógica em relação à sucção da bomba
      CADASTRO_SUCÇAO_INSUFICIENTE : Real;   // Cadastro de nível/pressão insuficiente
      CADASTRO_TEMPO_RESET : Time;   // Cadastro do tempo para resetar o alarme de Pressão Insuficiente
   END_VAR
   VAR_OUTPUT
      SUCÇÃO_OK : Bool;   // Sucção OK para operação
   END_VAR
   VAR
      SUCCAO_INSUFICIENTE : Bool;   // Sucção Insuficiente para operação
      RESET_ALARME : IEC_TIMER;   // Reset alarme de Sucção Insuficiente
   END_VAR
BEGIN

REGION Network 1: Set e Reset da Referência de Sucção insuficiente
   // Se nível for menor que a referência do Reservatório SUCÇÃO INSUFICIENTE,  bomba não pode ligar.
   // Caso o Nivel seja maior que a refêrencia então, após tempo cadastrado a bomba está habita para ligar
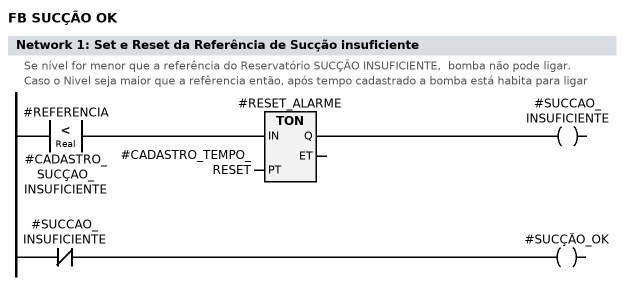
   #RESET_ALARME.TON(IN := #REFERENCIA < #CADASTRO_SUCÇAO_INSUFICIENTE, PT := #CADASTRO_TEMPO_RESET);
   #SUCCAO_INSUFICIENTE := #RESET_ALARME.Q;
   #SUCÇÃO_OK := NOT #SUCCAO_INSUFICIENTE;
END_REGION
END_FUNCTION_BLOCK

FUNCTION_BLOCK "FB VALVULA"   // FB17, LAD
{ S7_Optimized_Access := 'TRUE' }
VERSION : 0.1
// Network 1: Gerenciamento Status Válvula
// Network 2: Recebimento dos sinais de entrada (Sinais de campo e comandos)
// Network 3: MODO MANUAL: Conjunto de condições para ligar e desligar
// Network 4: MODO AUTOMÁTICO: Conjunto de condições para ligar e desligar
// Network 5: FALHA: Condicionamento de falha
// Network 6: LIGA BOMBA: Validando intertravamentos para ligar
// Network 7: ABRE VÁLVULA: Validando intertravamentos para abrir
   VAR_INPUT
      INPUT_ABERTA : Bool;   // 1 = Sinal elétrico de campo indicando válvula aberta
      INPUT_FECHADA : Bool;   // 1 = Sinal elétrico de campo indicando válvula fechada
      INPUT_FALHA : Bool;   // 0 = Sinal elétrico de campo indicando válvula em falha
      INPUT_LOCAL : Bool;   // 1 = Sinal elétrico de campo indicando válvula em modo local
      INPUT_REMOTO : Bool;   // 1 = Sinal elétrico de campo indicando válvula em modo remoto
      INPUT_FALHA_PROFINET : Bool;   // 1 = Indica falta de comunicação PROFINET com o equipamento
      INPUT_LIGA_AUTO : Bool;   // 1= indica que o processo pode ser ligado remoto manual
      PARAMETRO_ABRE : Bool;   // Parâmetro utilizado para abrir a válvula em modo automático
      PARAMETRO_FECHA : Bool;   // Parâmetro utilizado para fechar a válvula em modo automático
      CMD_ABRE : Bool;   // Comando enviado da IHM/SCADA para abrir a válvula
      CMD_MANUTEN : Bool;   // Comando enviado da IHM/SCADA para colocar a válvula em Modo de Manutenção
      CMD_MODO : Bool;   // Comando enviado da IHM/SCADA para colocar a bomba em (0 = Modo Manual, 1 = Modo Automático)
   END_VAR
   VAR_OUTPUT
      STATUS_VALV : Byte;   // 0 = FECHADA; 1 = ABERTA; 2 = FALHA
      ABRE_VALVULA : Bool;   // Saída acionada para abrir a válvula remotamente
      FECHA_VALVULA : Bool;   // Saída acionada para fechar a válvula remotamente
      REMOTO_MAN : Bool;   // Modo de Operação Remoto Manual
      REMOTO_AUTO : Bool;   // Modo de Operação Remoto Automático
      LOCAL_MAN : Bool;   // Modo de Operação Local Manual
   END_VAR
   VAR
      MANUTEN : Bool;   // Variável local para Indicar bomba em Modo Manutenção
      REMOTO : Bool;   // Variável local para indicar Modo Remoto
      FALHA : Bool;   // Variável local para Válvula em Falha
      ABRE_REM_MAN : Bool;   // Variável local para Acionamento Remoto Manual
      ABRE_REM_AUTO : Bool;   // Variável local para Acionamento Remoto Automático
   END_VAR
   VAR_TEMP   // added for the SCL form of the ladder/FBD networks
      _w1 : Bool;
   END_VAR
BEGIN

REGION Network 1: Gerenciamento Status Válvula
   // INPUT_ABERTA = Entrada de sinal de Válvula Aberta
   // INPUT_FECHADA = Entrada de sinal de Válvula Fechada
   // INPUT_FALHA = Entrada de sinal de Válvula em Falha
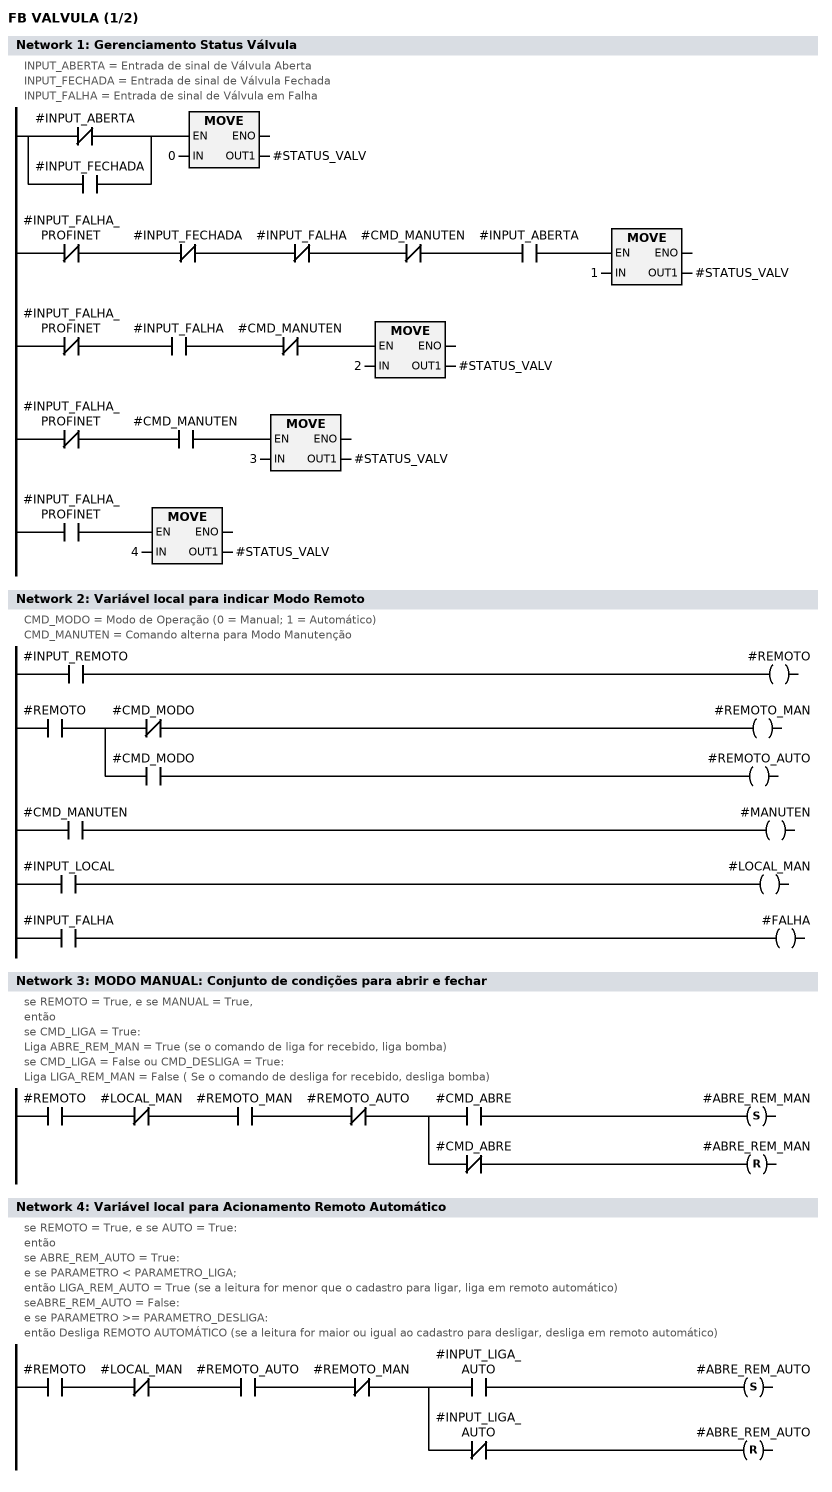
   RUNG wire#powerrail
      I_Contact( #INPUT_ABERTA )
      wire#w1
      Move(in := 0, out1 => #STATUS_VALV)
   END_RUNG
   RUNG wire#powerrail
      Contact( #INPUT_FECHADA )
   END_RUNG wire#w1
   RUNG wire#powerrail
      I_Contact( #INPUT_FALHA_PROFINET )
      I_Contact( #INPUT_FECHADA )
      I_Contact( #INPUT_FALHA )
      I_Contact( #CMD_MANUTEN )
      Contact( #INPUT_ABERTA )
      Move(in := 1, out1 => #STATUS_VALV)
   END_RUNG
   RUNG wire#powerrail
      I_Contact( #INPUT_FALHA_PROFINET )
      Contact( #INPUT_FALHA )
      I_Contact( #CMD_MANUTEN )
      Move(in := 2, out1 => #STATUS_VALV)
   END_RUNG
   RUNG wire#powerrail
      I_Contact( #INPUT_FALHA_PROFINET )
      Contact( #CMD_MANUTEN )
      Move(in := 3, out1 => #STATUS_VALV)
   END_RUNG
   RUNG wire#powerrail
      Contact( #INPUT_FALHA_PROFINET )
      Move(in := 4, out1 => #STATUS_VALV)
   END_RUNG
   // the same network as SCL:
   IF NOT #INPUT_ABERTA OR #INPUT_FECHADA THEN #STATUS_VALV := 0; END_IF;
   IF NOT #INPUT_FALHA_PROFINET AND NOT #INPUT_FECHADA AND NOT #INPUT_FALHA AND NOT #CMD_MANUTEN AND #INPUT_ABERTA THEN
       #STATUS_VALV := 1;
   END_IF;
   IF NOT #INPUT_FALHA_PROFINET AND #INPUT_FALHA AND NOT #CMD_MANUTEN THEN #STATUS_VALV := 2; END_IF;
   IF NOT #INPUT_FALHA_PROFINET AND #CMD_MANUTEN THEN #STATUS_VALV := 3; END_IF;
   IF #INPUT_FALHA_PROFINET THEN #STATUS_VALV := 4; END_IF;
END_REGION

REGION Network 2: Variável local para indicar Modo Remoto
   // CMD_MODO = Modo de Operação (0 = Manual; 1 = Automático)
   // CMD_MANUTEN = Comando alterna para Modo Manutenção
   RUNG wire#powerrail
      Contact( #INPUT_REMOTO )
      Coil( #REMOTO )
   END_RUNG
   RUNG wire#powerrail
      Contact( #REMOTO )
      wire#w1
      I_Contact( #CMD_MODO )
      Coil( #REMOTO_MAN )
   END_RUNG
   RUNG wire#w1
      Contact( #CMD_MODO )
      Coil( #REMOTO_AUTO )
   END_RUNG
   RUNG wire#powerrail
      Contact( #CMD_MANUTEN )
      Coil( #MANUTEN )
   END_RUNG
   RUNG wire#powerrail
      Contact( #INPUT_LOCAL )
      Coil( #LOCAL_MAN )
   END_RUNG
   RUNG wire#powerrail
      Contact( #INPUT_FALHA )
      Coil( #FALHA )
   END_RUNG
   // the same network as SCL:
   #REMOTO := #INPUT_REMOTO;
   #REMOTO_MAN := #REMOTO AND NOT #CMD_MODO;
   #REMOTO_AUTO := #REMOTO AND #CMD_MODO;
   #MANUTEN := #CMD_MANUTEN;
   #LOCAL_MAN := #INPUT_LOCAL;
   #FALHA := #INPUT_FALHA;
END_REGION

REGION Network 3: MODO MANUAL: Conjunto de condições para abrir e fechar
   // se REMOTO = True, e se MANUAL = True,
   // 
   // então
   // se CMD_LIGA = True: 
   // Liga ABRE_REM_MAN = True (se o comando de liga for recebido, liga bomba)
   // 
   // se CMD_LIGA = False ou CMD_DESLIGA = True:
   // Liga LIGA_REM_MAN = False ( Se o comando de desliga for recebido, desliga bomba)
   RUNG wire#powerrail
      Contact( #REMOTO )
      I_Contact( #LOCAL_MAN )
      Contact( #REMOTO_MAN )
      I_Contact( #REMOTO_AUTO )
      wire#w1
      Contact( #CMD_ABRE )
      S_Coil( #ABRE_REM_MAN )
   END_RUNG
   RUNG wire#w1
      I_Contact( #CMD_ABRE )
      R_Coil( #ABRE_REM_MAN )
   END_RUNG
   // the same network as SCL:
   #_w1 := #REMOTO AND NOT #LOCAL_MAN AND #REMOTO_MAN AND NOT #REMOTO_AUTO;
   IF #_w1 AND #CMD_ABRE THEN #ABRE_REM_MAN := TRUE; END_IF;
   IF #_w1 AND NOT #CMD_ABRE THEN #ABRE_REM_MAN := FALSE; END_IF;
END_REGION

REGION Network 4: Variável local para Acionamento Remoto Automático
   // se REMOTO = True, e se AUTO = True:
   // 
   // então
   // se ABRE_REM_AUTO = True:
   // e se PARAMETRO < PARAMETRO_LIGA;
   // então LIGA_REM_AUTO = True (se a leitura for menor que o cadastro para ligar, liga em remoto automático)
   // 
   // seABRE_REM_AUTO = False:
   // e se PARAMETRO >= PARAMETRO_DESLIGA:
   // então Desliga REMOTO AUTOMÁTICO (se a leitura for maior ou igual ao cadastro para desligar, desliga em remoto automático)
   RUNG wire#powerrail
      Contact( #REMOTO )
      I_Contact( #LOCAL_MAN )
      Contact( #REMOTO_AUTO )
      I_Contact( #REMOTO_MAN )
      wire#w1
      Contact( #INPUT_LIGA_AUTO )
      S_Coil( #ABRE_REM_AUTO )
   END_RUNG
   RUNG wire#w1
      I_Contact( #INPUT_LIGA_AUTO )
      R_Coil( #ABRE_REM_AUTO )
   END_RUNG
   // the same network as SCL:
   #_w1 := #REMOTO AND NOT #LOCAL_MAN AND #REMOTO_AUTO AND NOT #REMOTO_MAN;
   IF #_w1 AND #INPUT_LIGA_AUTO THEN #ABRE_REM_AUTO := TRUE; END_IF;
   IF #_w1 AND NOT #INPUT_LIGA_AUTO THEN #ABRE_REM_AUTO := FALSE; END_IF;
END_REGION

REGION Network 5: FALHA: Condicionamento de falha
   // se FALHA = False;
   // 
   // então
   // ABRE_REM_AUTO = False (Reseta Liga Remoto Automático)
   // ABRE_REM_MAN = False (Reseta Liga Remoto Manual)
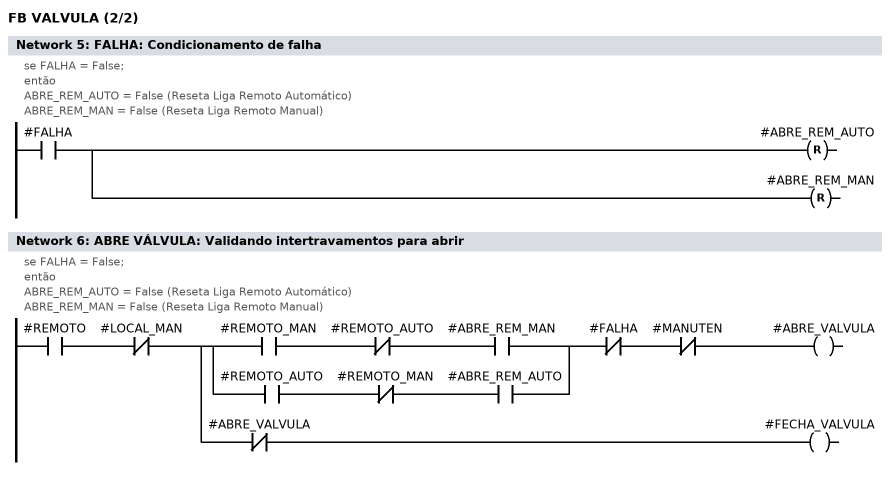
   RUNG wire#powerrail
      Contact( #FALHA )
      wire#w1
      R_Coil( #ABRE_REM_AUTO )
   END_RUNG
   RUNG wire#w1
      R_Coil( #ABRE_REM_MAN )
   END_RUNG
   // the same network as SCL:
   IF #FALHA THEN
       #ABRE_REM_AUTO := FALSE;
       #ABRE_REM_MAN := FALSE;
   END_IF;
END_REGION

REGION Network 6: ABRE VÁLVULA: Validando intertravamentos para abrir
   // se FALHA = False;
   // 
   // então
   // ABRE_REM_AUTO = False (Reseta Liga Remoto Automático)
   // ABRE_REM_MAN = False (Reseta Liga Remoto Manual)
   RUNG wire#powerrail
      Contact( #REMOTO )
      I_Contact( #LOCAL_MAN )
      wire#w1
      Contact( #REMOTO_MAN )
      I_Contact( #REMOTO_AUTO )
      Contact( #ABRE_REM_MAN )
      wire#w2
      I_Contact( #FALHA )
      I_Contact( #MANUTEN )
      Coil( #ABRE_VALVULA )
   END_RUNG
   RUNG wire#w1
      Contact( #REMOTO_AUTO )
      I_Contact( #REMOTO_MAN )
      Contact( #ABRE_REM_AUTO )
   END_RUNG wire#w2
   RUNG wire#w1
      I_Contact( #ABRE_VALVULA )
      Coil( #FECHA_VALVULA )
   END_RUNG
   // the same network as SCL:
   #_w1 := #REMOTO AND NOT #LOCAL_MAN;
   #ABRE_VALVULA := #_w1 AND ((#REMOTO_MAN AND NOT #REMOTO_AUTO AND #ABRE_REM_MAN) OR (#REMOTO_AUTO AND NOT #REMOTO_MAN AND #ABRE_REM_AUTO)) AND NOT #FALHA AND NOT #MANUTEN;
   #FECHA_VALVULA := #_w1 AND NOT #ABRE_VALVULA;
END_REGION
END_FUNCTION_BLOCK

FUNCTION_BLOCK "FB INTERTRAVAMENTO_PAINEL"   // FB27, SCL
{ S7_Optimized_Access := 'TRUE' }
VERSION : 0.1
   VAR_INPUT
      INPUT_BT_EMERGENCIA : Bool;
      INPUT_DISJUNTOR : Bool;
      INPUT_FONTE1 : Bool;
      INPUT_FONTE2 : Bool;
      INPUT_RELE_FALTA : Bool;
      INPUT_CONDICAO : Bool;
      INPUT_TESTE : Bool;
   END_VAR
   VAR_OUTPUT
      OUTPUT_PAINEL_OK : Bool;
   END_VAR
BEGIN

   IF ((#INPUT_BT_EMERGENCIA AND // Supondo que BT_EMERGENCIA é True quando ñ ATUADO
         NOT #INPUT_DISJUNTOR AND
         #INPUT_FONTE1 AND
         #INPUT_FONTE2 AND
         #INPUT_RELE_FALTA AND // Supondo que RELE_FALTA é True quando ñ ATUADO
         #INPUT_CONDICAO) 
      OR
      #INPUT_TESTE) THEN // teste força a saída 
   #OUTPUT_PAINEL_OK := TRUE;
   ELSE
       #OUTPUT_PAINEL_OK := FALSE;
   END_IF;
END_FUNCTION_BLOCK

// folder: 1. FB Bilbiotecas/1.1 Acionamento/1.1.1 Inversores

FUNCTION_BLOCK "FB AFERIÇÃO INVERSORES"   // FB2, LAD
{ S7_Optimized_Access := 'TRUE' }
VERSION : 0.1
// Os sinais de campo são recebidos em corrente (4-20mA) e representados pelo fundo de escala do CLP. Este bloco faz a conversão do sinal para a leitura real da medição.
// 
// Network 1: Ajuste do fundo de escala aos parâmetros de aferição
// Network 2: Cálculo da equação da reta para definir a leitura atual da entrada analógica
// Network 3: Setando o alarme SEM 4mA na entrada digital caso seja rompida
   VAR_INPUT
      ANALOG_IN_4a20mA : Int;   // Entrada do sinal analógico
      Y1_CONFIG : Int;   // Fundo de escala mínimo para o CLP
      Y2_CONFIG : Int;   // Fundo de escala máximo para o CLP
      X1_CONFIG : Int;   // Fundo de escala mínimo para o equipamento
      X2_CONFIG : Int;   // Fundo de escala máximo para o equipamento
      COMANDO : Int;   // Comando enviado da IHM/SCADA para aferir determinado equipamento
      COMANDO_VALOR : Int;   // Valor comparativo para executar o Bloco FB
      GRANDEZA_MAX : Int;   // Referência a grandeza maxima no qual o bloco vai utilizar para fazer a curva da reta
   END_VAR
   VAR_OUTPUT
      ANALOG_OUT_4a20mA : Real;   // Saída do sinal analógico já aferido
      ALARME_SEM_4mA : Bool;   // 1 = Entrada sem 4mA, indicando erro; 0 = Entrada OK
      RANGE_MIN_CADASTRADO : Int;   // Valor do cadastro máximo armazenado para visualizar na IHM
      RANGE_MAX_CADASTRADO : Int;   // Valor do cadastro mínimo armazenado para visualizar na IHM
   END_VAR
   VAR
      ANALOG_IN_LIMITED : Int;   // Tratamento de erro do sinal analógico para capturar apenas leituras que estão dentro do range do CLP
      ANALOG_IN_LIMITED_REAL : UInt;   // Saída do sinal ajustado conforme a grandeza máxima
      STATIC_X1 : UInt;   // Fundo de escala mínimo para o equipamento (Instanciado no FB)
      STATIC_X2 : UInt;   // Fundo de escala máximo para o equipamento (Instanciado no FB)
      STATIC_Y1 : UInt;   // Fundo de escala mínimo para o CLP (Instanciado no FB)
      STATIC_Y2 : UInt;   // Fundo de escala máximo para o CLP (Instanciado no FB)
      STATIC_GRANDEZA_MAX : UInt;   // Grandeza máxima do equipamento
      AJUSTAR_CURVA : Bool;   // Memória para mover as entradas às instâncias
      PONTO_ZERO : Int;   // Range mínimo do equipamento quando é diferente de 0
      ALARME_RESET : TOF_TIME;   // Reset do alarme Sem 4mA ao estabilizar o sinal
      PULSO_AJUSTAR : Bool;   // Pulso para realizar a aferição da curva
   END_VAR
   VAR_TEMP   // added for the SCL form of the ladder/FBD networks
      _w1 : Bool;
   END_VAR
BEGIN

REGION Network 1: Ajuste do fundo de escala aos parâmetros de aferição
   // X1_CONFIG = Fundo de escala mínimo para o equipamento
   // X2_CONFIG = Fundo de escala máximo para o equipamento
   // Y1_CONFIG = Fundo de escala mínimo para o CLP
   // Y2_CONFIG = Fundo de escala máximo para o CLP
   // GRANDEZA_MAX = Referência a grandeza maxima no qual o bloco vai utilizar para fazer a curva da reta
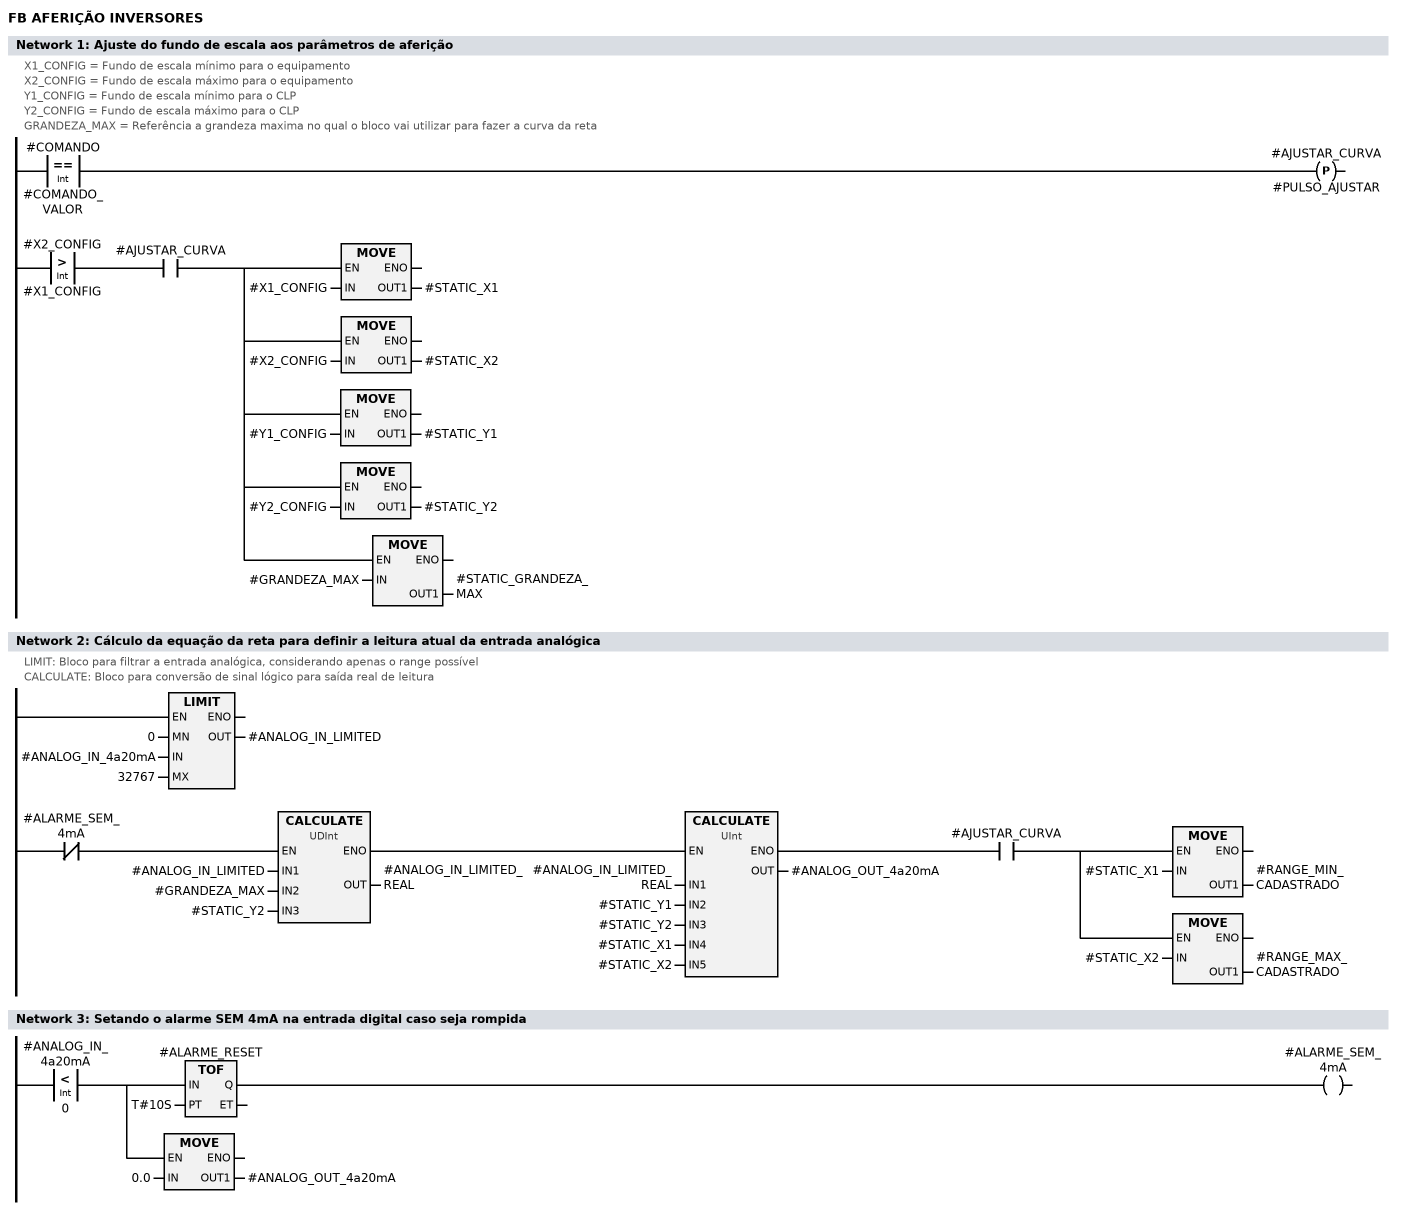
   #_w1 := #COMANDO = #COMANDO_VALOR;
   #AJUSTAR_CURVA := #_w1 AND NOT #PULSO_AJUSTAR;   // rising edge
   #PULSO_AJUSTAR := #_w1;
   IF (#X2_CONFIG > #X1_CONFIG) AND #AJUSTAR_CURVA THEN
       #STATIC_X1 := #X1_CONFIG;
       #STATIC_X2 := #X2_CONFIG;
       #STATIC_Y1 := #Y1_CONFIG;
       #STATIC_Y2 := #Y2_CONFIG;
       #STATIC_GRANDEZA_MAX := #GRANDEZA_MAX;
   END_IF;
END_REGION

REGION Network 2: Cálculo da equação da reta para definir a leitura atual da entrada analógica
   // LIMIT: Bloco para filtrar a entrada analógica, considerando apenas o range possível
   // CALCULATE: Bloco para conversão de sinal lógico para saída real de leitura
   #ANALOG_IN_LIMITED := LIMIT(MN := 0, IN := #ANALOG_IN_4a20mA, MX := 32767);
   IF NOT #ALARME_SEM_4mA THEN
       #ANALOG_IN_LIMITED_REAL := #ANALOG_IN_LIMITED * #STATIC_Y2 / #GRANDEZA_MAX;
       #ANALOG_OUT_4a20mA := (#ANALOG_IN_LIMITED_REAL - #STATIC_Y1) * (#STATIC_X2 - #STATIC_X1) / (#STATIC_Y2 - #STATIC_Y1);
   END_IF;
   IF NOT #ALARME_SEM_4mA AND #AJUSTAR_CURVA THEN
       #RANGE_MIN_CADASTRADO := #STATIC_X1;
       #RANGE_MAX_CADASTRADO := #STATIC_X2;
   END_IF;
END_REGION

REGION Network 3: Setando o alarme SEM 4mA na entrada digital caso seja rompida
   #_w1 := #ANALOG_IN_4a20mA < 0;
   #ALARME_RESET(IN := #_w1, PT := T#10S);   // TOF
   #ALARME_SEM_4mA := #ALARME_RESET.Q;
   IF #_w1 THEN #ANALOG_OUT_4a20mA := 0.0; END_IF;
END_REGION
END_FUNCTION_BLOCK

FUNCTION_BLOCK "FB STATUS ECSX"   // FB12, LAD
TITLE = Function Block STATUS ECSX - Status dos exaustores (ECS1 - ECS2 - ECS3)
{ S7_Optimized_Access := 'TRUE' }
VERSION : 0.1
// Sinais de status (ligado e falha) recebidos de campo
   VAR_INPUT
      INPUT_LIGADO : Bool;   // Entrada do sinal de Motor/Bomba ligado
      INPUT_FALHA : Bool;   // Entrada do sinal de falha instanciado na Network 1
      INPUT_MANUTEN : Bool;   // Entrada do sinal de manutenção instanciado na Network 1
      INPUT_FALHA_PROFINET : Bool;   // 1 = Indica falta de comunicação PROFINET com o equipamento
   END_VAR
   VAR_OUTPUT
      STATUS_MOTOR : Byte;   // Indicador de Status do exaustor
   END_VAR
BEGIN

REGION Network 1: Acionamento do status ligado
   // INUPT_LIGADO = TRUE: Exaustor ligado
   // INPUT_FALHA = TRUE: Exaustor em falha
   // INPUT_FALHA_PROFINET = TRUE: Sem Comunicação PROFINET
   // INPUT_MANUTEN = TRUE: Motor/Exaustor em manutenção
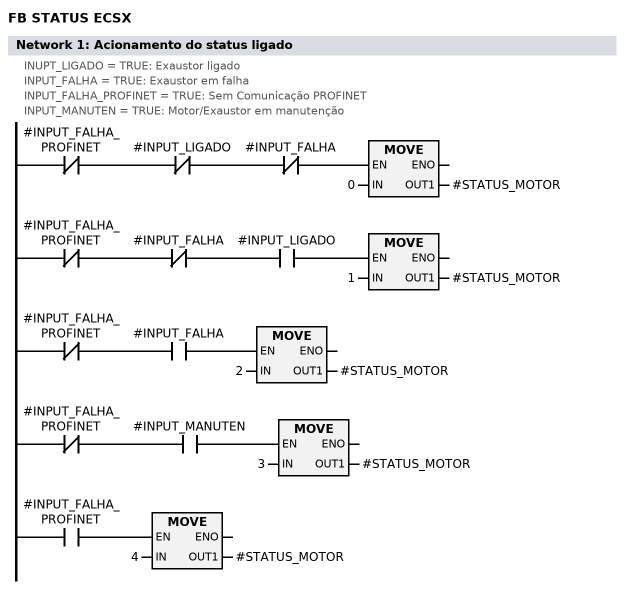
   RUNG wire#powerrail
      I_Contact( #INPUT_FALHA_PROFINET )
      I_Contact( #INPUT_LIGADO )
      I_Contact( #INPUT_FALHA )
      Move(in := 0, out1 => #STATUS_MOTOR)
   END_RUNG
   RUNG wire#powerrail
      I_Contact( #INPUT_FALHA_PROFINET )
      I_Contact( #INPUT_FALHA )
      Contact( #INPUT_LIGADO )
      Move(in := 1, out1 => #STATUS_MOTOR)
   END_RUNG
   RUNG wire#powerrail
      I_Contact( #INPUT_FALHA_PROFINET )
      Contact( #INPUT_FALHA )
      Move(in := 2, out1 => #STATUS_MOTOR)
   END_RUNG
   RUNG wire#powerrail
      I_Contact( #INPUT_FALHA_PROFINET )
      Contact( #INPUT_MANUTEN )
      Move(in := 3, out1 => #STATUS_MOTOR)
   END_RUNG
   RUNG wire#powerrail
      Contact( #INPUT_FALHA_PROFINET )
      Move(in := 4, out1 => #STATUS_MOTOR)
   END_RUNG
   // the same network as SCL:
   IF NOT #INPUT_FALHA_PROFINET AND NOT #INPUT_LIGADO AND NOT #INPUT_FALHA THEN #STATUS_MOTOR := 0; END_IF;
   IF NOT #INPUT_FALHA_PROFINET AND NOT #INPUT_FALHA AND #INPUT_LIGADO THEN #STATUS_MOTOR := 1; END_IF;
   IF NOT #INPUT_FALHA_PROFINET AND #INPUT_FALHA THEN #STATUS_MOTOR := 2; END_IF;
   IF NOT #INPUT_FALHA_PROFINET AND #INPUT_MANUTEN THEN #STATUS_MOTOR := 3; END_IF;
   IF #INPUT_FALHA_PROFINET THEN #STATUS_MOTOR := 4; END_IF;
END_REGION
END_FUNCTION_BLOCK

FUNCTION_BLOCK "FB INVERSOR SIEMENS"   // FB20, LAD
{ S7_Optimized_Access := 'TRUE' }
VERSION : 0.1
   VAR_INPUT
      RPM_min_Driver : Int;
      RPM_Max_Driver : Int;
      Setpoint_Velocidade : Int;
   END_VAR
   VAR_OUTPUT
      Telegram_Out_Velocidade : Int;
   END_VAR
   VAR_TEMP
      Aux_Velocidade : Real;
   END_VAR
BEGIN

REGION Network 1: Controle Velocidade
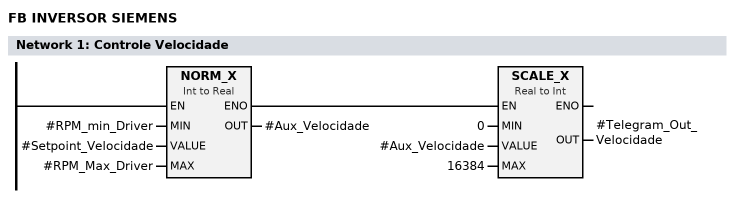
   RUNG wire#powerrail
      { S7_Templates := "[SrcType := Int, DestType := Real]" } Normalize(min := #RPM_min_Driver, value := #Setpoint_Velocidade, max := #RPM_Max_Driver, out => #Aux_Velocidade)
      { S7_Templates := "[SrcType := Real, DestType := Int]" } Scale(min := 0, value := #Aux_Velocidade, max := 16384, out => #Telegram_Out_Velocidade)
   END_RUNG
   // the same network as SCL:
   #Aux_Velocidade := NORM_X(MIN := #RPM_min_Driver, VALUE := #Setpoint_Velocidade, MAX := #RPM_Max_Driver);
   #Telegram_Out_Velocidade := SCALE_X(MIN := 0, VALUE := #Aux_Velocidade, MAX := 16384);
END_REGION
END_FUNCTION_BLOCK

FUNCTION_BLOCK "SINA_SPEED_TLG20"   // FB38003, SCL
TITLE = Speed control S7 to SINAMICS using Standardtelegram 20
{ S7_Optimized_Access := 'TRUE' }
AUTHOR : SIEMENS
FAMILY : DRIVES
NAME : SINA_SPD_TLG20
VERSION : 1.0
// The function block SINA_SPEED_TLG20 controls a SINAMICS drive using standard telegram 20
   VAR_INPUT
      enableAxis : Bool;   // 0 -> 1 = Enable the drive (OFF2 / OFF 3 are 1 in default status) (OFF1 = 0->1)
      ackError : Bool;   // 0 -> 1 = Acknowledge drive error
      speedSp : Real;   // Speed setpoint [rpm]
      selectCDS : USInt;   // Selection of the Command Data Set (0 = CDS0, 1 = CDS1)
      refSpeed : Real;   // Reference speed [p2000] in [rpm]
      refCurrent : Real;   // Reference current [p2002] in [Aeff]
      refTorque : Real;   // Reference torque [p2003] in [Nm]
      refPower : Real;   // Reference power [r2005] in [kW]
      configAxis : Word := 16#003F;   // binary programmed input to control all functions in the telegram without its own function block input
      HWIDSTW : HW_IO;   // Hardware Identifer set point slot
      HWIDZSW : HW_IO;   // Hardware Identifer actual value slot
   END_VAR
   VAR_OUTPUT
      axisEnabled : Bool;   // 1 = Drive is enabled
      lockout : Bool;   // 1 = Drive lockout active
      actCDS : USInt;   // Active Command Data Set (0 = CDS0, 1 = CDS1)
      actSpeed : Real;   // Smoothed actual speed in [1/min]
      actCurrent : Real;   // Smoothed current actual in [Arms]
      actTorque : Real;   // Actual smoothed torque in [Nm]
      actPower : Real;   // Actual smoothed active power in [kW]
      faultVIKNAMUR : Word;   // Fault word according to the VIK-NAMUR defintion
      error : Bool;   // 1 = Error (FB and Infeed)
      status : Int;   // Status output (7002 = FB in operation; 7xxx = warning; 8xxx = error description - read the manual)
      diagId : Int;   // Error codes of the system function blocks DPWR / DPRD_DAT
   END_VAR
   VAR_TEMP
      tempSpeed : Real;   // Speed setpoint in percent
      tempRefValueInvalid : Bool;   // At least one reference value is 0 or < 0
      tempSendBuf : Array[0..1] of Word;   // Send buffer
      tempRecvBuf : Array[0..5] of Word;   // Receive buffer
   END_VAR
   VAR CONSTANT
      NORMALIZATION_VALUE : Int := 16#4000;   // Used to calculate the Real values
      MAX_INT : Int := 16#7FFF;
      MIN_INT : Int := 16#8000;
      REF_CURRRENT_INVALID : Int := 16#7010;   // RefCurrent input is 0 or < 0
      REF_TORQUE_INVALID : Int := 16#7011;   // RefTorque input is 0 or < 0
      REF_POWER_INVALID : Int := 16#7012;   // RefPower input is 0 or < 0
      REF_VALUES_INVALID : Int := 16#7013;   // Multiple reference values are 0 or < 0
      NO_ERROR : Int := 16#7002;   // No error
      ERROR_REF_SPEED_INVALID : Int := 16#8001;   // RefSpeed input is 0 or < 0
      ERROR_INVALID_CDS : Int := 16#8002;   // Invalid Command Data Set selected
      ERROR_DRIVE : Int := 16#8401;   // Drive error
      ERROR_LOCKOUT : Int := 16#8402;   // Drive lockout
      ERROR_DPREAD : Int := 16#8600;   // DPRD_DAT returned an error
      ERROR_DPWRITE : Int := 16#8601;   // DPWR_DAT returned an error
      ERROR_FAULT_WORD : Int := 16#8700;   // faultVIKNAMUR is not 0
      STW1 : USInt := 0;
      ZSW1 : USInt := 0;
      NSOLL_A : USInt := 1;
   END_VAR
BEGIN
   //=============================================================================
   //SIEMENS AG
   //(c)Copyright 2019 All Rights Reserved
   //-----------------------------------------------------------------------------
   // Library:       LSINAExt
   // Tested with:   SIMATIC S7 CPU 1513-1 PN V2.5
   // Engineering:   TIA Portal V15
   // Restrictions:  -
   // Requirements:  S7-1200 / S7-1500
   // Functionality: cyclic communication between a SINAMICS a PLC.
   //                If in HWConfig standard telegram 20 are projected 2 PZD-words are exchanged
   //                in every bus cycle.
   //                The parametrisation of these words is described in the manual of the
   //                SINAMICS
   //-----------------------------------------------------------------------------
   //Change log table:
   //Version  Date       Expert in charge Changes applied
   //01.00.00 11.02.2019 (AS) First released version
   //=============================================================================

   // Prepare PZD1 (STW1)
   #tempSendBuf[#STW1].%X0 := #enableAxis;
   #tempSendBuf[#STW1].%X7 := #ackError;
   #tempSendBuf[#STW1].%X1 := #configAxis.%X0;
   #tempSendBuf[#STW1].%X2 := #configAxis.%X1;
   #tempSendBuf[#STW1].%X3 := #configAxis.%X2;
   #tempSendBuf[#STW1].%X4 := #configAxis.%X3;
   #tempSendBuf[#STW1].%X5 := #configAxis.%X4;
   #tempSendBuf[#STW1].%X6 := #configAxis.%X5;
   #tempSendBuf[#STW1].%X11 := #configAxis.%X6;
   #tempSendBuf[#STW1].%X15 := #selectCDS = 1; // true = CDS0, false = CDS1
   #tempSendBuf[#STW1].%X10 := TRUE; // control by PLC
   #tempSendBuf[#STW1].%X13 := FALSE; // STW1.X13 not used in Telegram 20
   #tempSendBuf[#STW1].%X14 := FALSE; // STW1.X14 not used in Telegram 20

   // Check CDS index
   IF (#selectCDS < 0)
       OR (#selectCDS > 1)
   THEN
       #error := TRUE;
       #status := #ERROR_INVALID_CDS;
       #tempSendBuf[#STW1].%X0 := FALSE; // disable axis
   END_IF;

   // Speed
   IF #refSpeed > 0 THEN
       #tempSpeed := #speedSp * (#NORMALIZATION_VALUE / #refSpeed);
       // Limit REAL - Variable to INT - limits
       IF #tempSpeed > #MAX_INT
       THEN
           #tempSpeed := #MAX_INT;
       ELSIF #tempSpeed < #MIN_INT
       THEN
           #tempSpeed := #MIN_INT;
       ELSE
           ; // not needed
       END_IF;
       #tempSendBuf[#NSOLL_A] := INT_TO_WORD(REAL_TO_INT(#tempSpeed));
   ELSE
       #error := TRUE;
       #status := #ERROR_REF_SPEED_INVALID;
       #tempSendBuf[#NSOLL_A] := W#16#0;
   END_IF;

   // Send telegram to drive
   #diagId := DPWR_DAT(LADDR := #HWIDSTW,
                       RECORD := #tempSendBuf);

   // Error when writing the telegram
   IF #diagId <> 0 THEN
       #error := TRUE;
       #status := #ERROR_DPWRITE;

       // Reset outputs
       #actSpeed := 0.0;
       #actCurrent := 0.0;
       #actTorque := 0.0;
       #actPower := 0.0;
       #faultVIKNAMUR := W#16#0;

       RETURN;
   ELSE
       ;
   END_IF;

   // Receive telegram from drive
   #diagId := DPRD_DAT(LADDR := #HWIDZSW,
                       RECORD => #tempRecvBuf);

   // Error when reading the telegram
   IF #diagId <> 0 THEN
       #error := TRUE;
       #status := #ERROR_DPREAD;

       // Reset outputs
       #actSpeed := 0.0;
       #actCurrent := 0.0;
       #actTorque := 0.0;
       #actPower := 0.0;
       #faultVIKNAMUR := W#16#0;

       RETURN;
   ELSE
       ;
   END_IF;

   // Analyse ZSW1
   #axisEnabled := #tempRecvBuf[#ZSW1].%X2;
   #lockout := #tempRecvBuf[#ZSW1].%X6;
   #error := #tempRecvBuf[#ZSW1].%X3 OR #tempRecvBuf[#ZSW1].%X6;

   IF #tempRecvBuf[#ZSW1].%X3 THEN
       #status := #ERROR_DRIVE;
   ELSIF #tempRecvBuf[#ZSW1].%X6 THEN
       #status := #ERROR_LOCKOUT;
   ELSE
       #status := #NO_ERROR;
   END_IF;

   // Check CDS
   IF #tempRecvBuf[#ZSW1].%X15 THEN
       #actCDS := 1;
   ELSE
       #actCDS := 0;
   END_IF;

   //IF #actCDS <> #selectCDS THEN
   //  #error := TRUE;
   //  #status := #ERROR_INVALID_CDS;
   //END_IF;

   // Actual speed
   IF (#refSpeed <= 0)
       AND #enableAxis
   THEN
       #actSpeed := 0.0;
       #error := TRUE;
       #status := #ERROR_REF_SPEED_INVALID;
   ELSE
       #actSpeed := INT_TO_REAL(WORD_TO_INT(#tempRecvBuf[1])) / (#NORMALIZATION_VALUE / #refSpeed);
   END_IF;

   // Actual current
   IF (#refCurrent <= 0)
       AND #enableAxis
       AND NOT #error
   THEN
       #actCurrent := 0.0;

       IF #tempRefValueInvalid THEN
           #status := #REF_VALUES_INVALID;
       ELSE
           #status := #REF_CURRRENT_INVALID;
           #tempRefValueInvalid := TRUE;
       END_IF;
   ELSE
       #actCurrent := INT_TO_REAL(WORD_TO_INT(#tempRecvBuf[2])) / (#NORMALIZATION_VALUE / #refCurrent);
   END_IF;

   // Actual torque
   IF (#refTorque <= 0)
       AND #enableAxis
       AND NOT #error
   THEN
       #actTorque := 0.0;

       IF #tempRefValueInvalid THEN
           #status := #REF_VALUES_INVALID;
       ELSE
           #status := #REF_TORQUE_INVALID;
           #tempRefValueInvalid := TRUE;
       END_IF;
   ELSE
       #actTorque := INT_TO_REAL(WORD_TO_INT(#tempRecvBuf[3])) / (#NORMALIZATION_VALUE / #refTorque);
   END_IF;

   // Actual active power
   IF (#refPower <= 0)
       AND #enableAxis
       AND NOT #error
   THEN
       #actPower := 0.0;

       IF #tempRefValueInvalid THEN
           #status := #REF_VALUES_INVALID;
       ELSE
           #status := #REF_POWER_INVALID;
           #tempRefValueInvalid := TRUE;
       END_IF;
   ELSE
       #actPower := INT_TO_REAL(WORD_TO_INT(#tempRecvBuf[4])) / (#NORMALIZATION_VALUE / #refPower);
   END_IF;

   // VIKNAMUR fault word
   #faultVIKNAMUR := #tempRecvBuf[5];
   IF #faultVIKNAMUR <> 16#0000 THEN
       #error := TRUE;
       #status := #ERROR_FAULT_WORD;
   ELSE
       ;
   END_IF;
END_FUNCTION_BLOCK

// folder: 1. FB Bilbiotecas/1.3 Instrumentação

FUNCTION_BLOCK "FB AFERIÇÃO INSTRUMENTOS"   // FB4, LAD
{ S7_Optimized_Access := 'TRUE' }
VERSION : 0.1
// Os sinais de campo são recebidos em corrente (4-20mA) e representados pelo fundo de escala do CLP. Este bloco faz a conversão do sinal para a leitura real da medição.
// 
// Network 1: Ajuste do fundo de escala aos parâmetros de aferição
// Network 2: Cálculo da equação da reta para definir a leitura atual da entrada analógica
// Network 3: Setando o alarme SEM 4mA na entrada digital caso seja rompida
   VAR_INPUT
      ANALOG_IN_4a20mA : Int;   // Entrada do sinal analógico para aferição
      X1_CONFIG : Int;   // Entrada do fundo de escala mínimo para o CLP
      X2_CONFIG : Int;   // Entrada do fundo de escala máximo para o CLP
      Y1_CONFIG : Int;   // Entrada do fundo de escala mínimo para o equipamento
      Y2_CONFIG : Int;   // Entrada do fundo de escala máximo para o equipamento
      COMANDO : Int;   // Valor enviado da IHM/SCADA para selecionar o equipamento
      COMANDO_VALOR : Int;   // Valor fixo na entrada do bloco para comparação com o COMANDO
   END_VAR
   VAR_OUTPUT
      ANALOG_OUT_4a20mA : Real;   // Saída do sinal analógico já aferido
      ALARME_SEM_4mA : Bool;   // 1 = Entrada sem 4mA, indicando erro; 0 = Entrada OK
      RANGE_MIN_CADASTRADO : UInt;   // Valor do cadastro mínimo armazenado para visualizar na IHM
      RANGE_MAX_CADASTRADO : UInt;   // Valor do cadastro máximo armazenado para visualizar na IHM
   END_VAR
   VAR RETAIN
      ANALOG_IN_LIMITED : Int;   // Tratamento de erro do sinal analógico para capturar apenas leituras que estão dentro do range do CLP
      STATIC_X1 : UInt;   // Fundo de escala mínimo para o equipamento (Instanciado no FB)
      STATIC_X2 : UInt;   // Fundo de escala máximo para o equipamento (Instanciado no FB)
      STATIC_Y1 : UInt;   // Fundo de escala mínimo para o CLP (Instanciado no FB)
      STATIC_Y2 : UInt;   // Fundo de escala máximo para o CLP (Instanciado no FB)
      AJUSTAR_CURVA : Bool;   // Memória para mover as entradas às instâncias
      PONTO_ZERO : Int;   // Range mínimo do equipamento quando é diferente de 0
      ALARME_RESET : TON_TIME;   // Reset do alarme Sem 4mA ao estabilizar o sinal
      PULSO_AJUSTAR : Bool;   // Pulso para realizar a aferição da curva
   END_VAR
   VAR
      RANGE_MIN_SEM_4mA : Int;
   END_VAR
   VAR_TEMP
      CURVA_RESULT : UInt;   // Resultado da curva pré-seleção da unidade de saída
   END_VAR
   VAR_TEMP   // added for the SCL form of the ladder/FBD networks
      _w1 : Bool;
   END_VAR
BEGIN

REGION Network 1: Ajuste do fundo de escala aos parâmetros de aferição
   // X1_CONFIG = Fundo de escala mínimo para o equipamento
   // X2_CONFIG = Fundo de escala máximo para o equipamento
   // Y1_CONFIG = Fundo de escala mínimo para o CLP
   // Y2_CONFIG = Fundo de escala máximo para o CLP
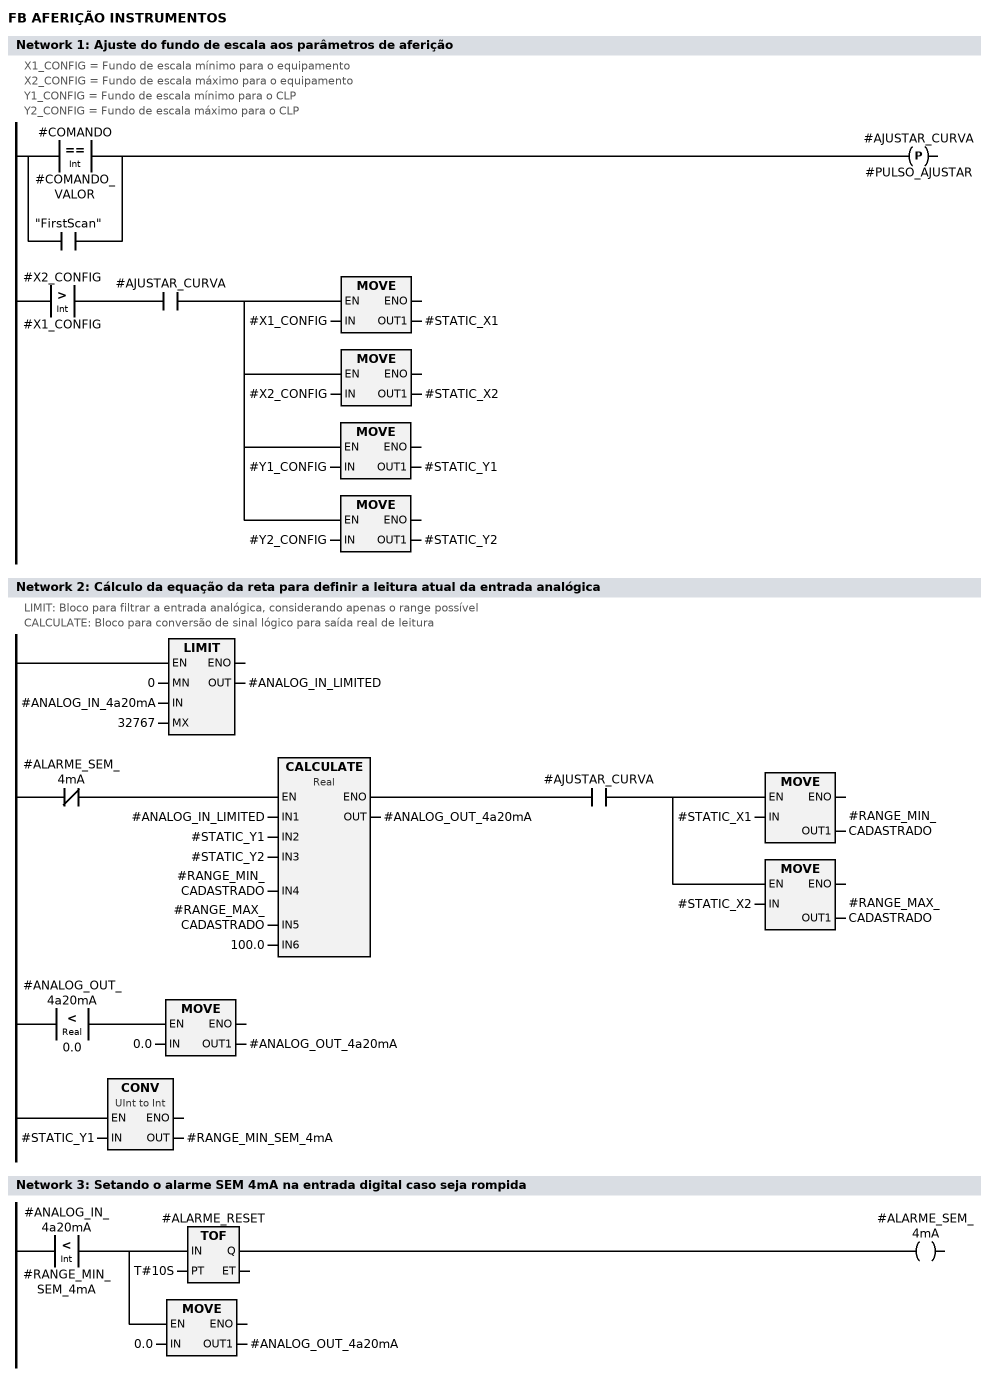
   #_w1 := (#COMANDO = #COMANDO_VALOR) OR "FirstScan";
   #AJUSTAR_CURVA := #_w1 AND NOT #PULSO_AJUSTAR;   // rising edge
   #PULSO_AJUSTAR := #_w1;
   IF (#X2_CONFIG > #X1_CONFIG) AND #AJUSTAR_CURVA THEN
       #STATIC_X1 := #X1_CONFIG;
       #STATIC_X2 := #X2_CONFIG;
       #STATIC_Y1 := #Y1_CONFIG;
       #STATIC_Y2 := #Y2_CONFIG;
   END_IF;
END_REGION

REGION Network 2: Cálculo da equação da reta para definir a leitura atual da entrada analógica
   // LIMIT: Bloco para filtrar a entrada analógica, considerando apenas o range possível
   // CALCULATE: Bloco para conversão de sinal lógico para saída real de leitura
   #ANALOG_IN_LIMITED := LIMIT(MN := 0, IN := #ANALOG_IN_4a20mA, MX := 32767);
   IF NOT #ALARME_SEM_4mA THEN
       #ANALOG_OUT_4a20mA := (((#ANALOG_IN_LIMITED - #STATIC_Y1) * (#RANGE_MAX_CADASTRADO - #RANGE_MIN_CADASTRADO)) / (#STATIC_Y2 - #STATIC_Y1))/100.0;
   END_IF;
   IF NOT #ALARME_SEM_4mA AND #AJUSTAR_CURVA THEN
       #RANGE_MIN_CADASTRADO := #STATIC_X1;
       #RANGE_MAX_CADASTRADO := #STATIC_X2;
   END_IF;
   IF #ANALOG_OUT_4a20mA < 0.0 THEN #ANALOG_OUT_4a20mA := 0.0; END_IF;
   #RANGE_MIN_SEM_4mA := UINT_TO_INT(#STATIC_Y1);
END_REGION

REGION Network 3: Setando o alarme SEM 4mA na entrada digital caso seja rompida
   #_w1 := #ANALOG_IN_4a20mA < #RANGE_MIN_SEM_4mA;
   #ALARME_RESET(IN := #_w1, PT := T#10S);   // TOF
   #ALARME_SEM_4mA := #ALARME_RESET.Q;
   IF #_w1 THEN #ANALOG_OUT_4a20mA := 0.0; END_IF;
END_REGION
END_FUNCTION_BLOCK

FUNCTION_BLOCK "FB SETPOINT ESCALONAMENTO"   // FB13, LAD
TITLE = Function Block SETPOINT L/H TO RPM - Bloco para escalonar o setpoint de uma unidade para rpm
{ S7_Optimized_Access := 'TRUE' }
VERSION : 0.1
// Network 1: Escalonamento dos ranges
   VAR_INPUT
      MAX_UNIT : Int;   // Unidade máxima para escalonamento
      MAX_RPM_TOTAL : Int;   // RPM total do equipamento
      MAX_RPM_IHM : Int;   // RPM máximo cadastrado pela IHM
      MIN_RPM_IHM : Int;   // RPM mínimo cadastrado pela IHM
   END_VAR
   VAR_OUTPUT
      SETPOINT_UNIT_OUT : Int;   // Setpoint da unidade convertida em rpm
      SETPOINT_UNIT_IN : Int;
   END_VAR
   VAR_IN_OUT
      SETPOINT : Int;   // Setpoint em unidade recebido da IHM
   END_VAR
   VAR RETAIN
      SETPOINT_MIN_UNIT : Int;   // Setpoint mínimo calculado de rpm para unidade
      SETPOINT_MAX_UNIT : Int;   // Setpoint máximo calculado de rpm para unidade
   END_VAR
BEGIN

REGION Network 1: Escalonamento dos ranges
   // MAX_RPM = RPM máximo cadastrado pela IHM
   // MIN_RPM = RPM mínimo cadastrado pela IHM
   // MAX_RPM_TOTAL = Limite físico máximo em rpm dos sopradores
   // MAX_UNIT = Pressão máxima dos sopradores
   // SETPOINT_RPM = Setpoint de milibar convertido em rpm
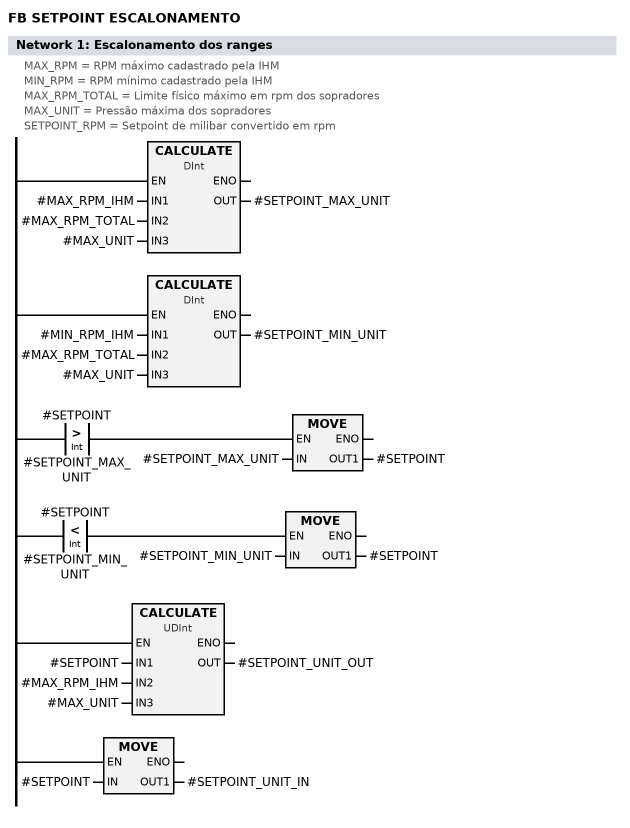
   RUNG wire#powerrail
      { S7_Templates := "SrcType := DInt"; S7_Expression := "(IN1*IN3) / IN2" } Calculate(in1 := #MAX_RPM_IHM, in2 := #MAX_RPM_TOTAL, in3 := #MAX_UNIT, out => #SETPOINT_MAX_UNIT)
   END_RUNG
   RUNG wire#powerrail
      { S7_Templates := "SrcType := DInt"; S7_Expression := "(IN1*IN3) / IN2" } Calculate(in1 := #MIN_RPM_IHM, in2 := #MAX_RPM_TOTAL, in3 := #MAX_UNIT, out => #SETPOINT_MIN_UNIT)
   END_RUNG
   RUNG wire#powerrail
      { S7_Templates := "SrcType := Int" } GT_Contact(in1 := #SETPOINT, in2 := #SETPOINT_MAX_UNIT)
      Move(in := #SETPOINT_MAX_UNIT, out1 => #SETPOINT)
   END_RUNG
   RUNG wire#powerrail
      { S7_Templates := "SrcType := Int" } LT_Contact(in1 := #SETPOINT, in2 := #SETPOINT_MIN_UNIT)
      Move(in := #SETPOINT_MIN_UNIT, out1 => #SETPOINT)
   END_RUNG
   RUNG wire#powerrail
      { S7_Templates := "SrcType := UDInt"; S7_Expression := "(IN1*IN2) / IN3" } Calculate(in1 := #SETPOINT, in2 := #MAX_RPM_IHM, in3 := #MAX_UNIT, out => #SETPOINT_UNIT_OUT)
   END_RUNG
   RUNG wire#powerrail
      Move(in := #SETPOINT, out1 => #SETPOINT_UNIT_IN)
   END_RUNG
   // the same network as SCL:
   #SETPOINT_MAX_UNIT := (#MAX_RPM_IHM*#MAX_UNIT) / #MAX_RPM_TOTAL;
   #SETPOINT_MIN_UNIT := (#MIN_RPM_IHM*#MAX_UNIT) / #MAX_RPM_TOTAL;
   IF #SETPOINT > #SETPOINT_MAX_UNIT THEN #SETPOINT := #SETPOINT_MAX_UNIT; END_IF;
   IF #SETPOINT < #SETPOINT_MIN_UNIT THEN #SETPOINT := #SETPOINT_MIN_UNIT; END_IF;
   #SETPOINT_UNIT_OUT := (#SETPOINT*#MAX_RPM_IHM) / #MAX_UNIT;
   #SETPOINT_UNIT_IN := #SETPOINT;
END_REGION
END_FUNCTION_BLOCK

FUNCTION_BLOCK "FB SETPOINT MANUAL"   // FB14, LAD
TITLE = Function Block FB SETPOINT_MANUAL
{ S7_Optimized_Access := 'TRUE' }
VERSION : 0.1
// Cálculo de conversão do valor setado, para escala do CLP.
   VAR_INPUT
      REMOTO : Bool;   // Recebe sinal de Remoto Manual
      COMANDO_VALOR : Int;   // Índice de comparação do bloco
      COMANDO : Int;   // Comando enviado via IHM/SCADA para definir min/max do range
      RANGE_MIN : Int;   // Valor mínimo do fundo de escala do equip, escrito via aferição
      RANGE_MAX : Int;   // Valor máximo do fundo de escala do equip, escrito via aferição
   END_VAR
   VAR_OUTPUT
      VALOR_SAIDA : Int;   // Valor de escrita no escravo.
      CADASTRO_VEL_MAX : Int;   // Cadastro da Velocidade Máxima via IHM
      CADASTRO_VEL_MIN : Int;   // Cadastro da Velocidade Mínima via IHM
   END_VAR
   VAR_IN_OUT
      SET_MANUAL : Int;   // Valor da grandeza a ser alcançado, escrita via aferição.
   END_VAR
   VAR RETAIN
      SETPOINT : Int;   // Setpoint de velocidade
      PULSE : Bool;
      PULSE_AUX : Bool;
   END_VAR
   VAR_TEMP   // added for the SCL form of the ladder/FBD networks
      _w1 : Bool;
   END_VAR
BEGIN

REGION Network 1: Cálculo Dosagem Manual
   // SET_MANUAL =  Valor da grandeza a ser alcançado, escrita via aferição.
   // RANGE_MAX   =  Valor máximo do fundo de escala do equip, escrita via aferição.
   // RANGE_MIN   =   Valor mínimo do fundo de escala do equip, escrita via aferição
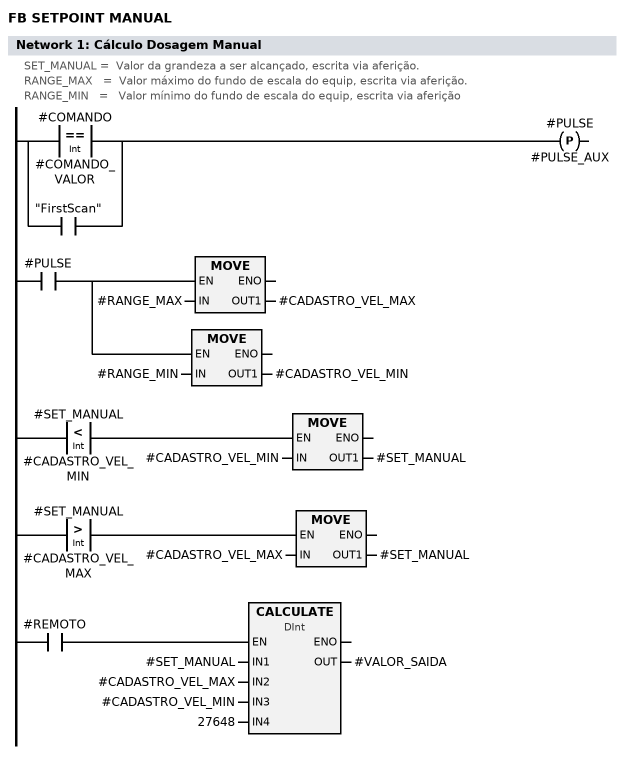
   #_w1 := (#COMANDO = #COMANDO_VALOR) OR "FirstScan";
   #PULSE := #_w1 AND NOT #PULSE_AUX;   // rising edge
   #PULSE_AUX := #_w1;
   IF #PULSE THEN
       #CADASTRO_VEL_MAX := #RANGE_MAX;
       #CADASTRO_VEL_MIN := #RANGE_MIN;
   END_IF;
   IF #SET_MANUAL < #CADASTRO_VEL_MIN THEN #SET_MANUAL := #CADASTRO_VEL_MIN; END_IF;
   IF #SET_MANUAL > #CADASTRO_VEL_MAX THEN #SET_MANUAL := #CADASTRO_VEL_MAX; END_IF;
   IF #REMOTO THEN
       #VALOR_SAIDA := ((#SET_MANUAL*27648) / (#CADASTRO_VEL_MAX-#CADASTRO_VEL_MIN)) - ((#CADASTRO_VEL_MIN*27648) / (#CADASTRO_VEL_MAX-#CADASTRO_VEL_MIN));
   END_IF;
END_REGION
END_FUNCTION_BLOCK

FUNCTION_BLOCK "FB FILTRO DE AMOSTRAGEM  ANALÍTICA"   // FB24, LAD
{ S7_Optimized_Access := 'TRUE' }
VERSION : 0.1
   VAR_INPUT
      INPUT_SENSOR : Int;
   END_VAR
   VAR_OUTPUT
      OUTPUT_SENSOR : Int;
   END_VAR
   VAR
      INDEX_AMOSTRAGEM : Int;
      AUX_1 : Int;
      AUX_2 : Int;
      AUX_3 : Int;
      AUX_4 : Int;
      AUX_5 : Int;
      AUX_6 : Int;
      AUX_7 : Int;
      AUX_8 : Int;
      AUX_9 : Int;
      AUX_10 : Bool;
      AUX_11 : Int;
   END_VAR
   VAR_TEMP   // added for the SCL form of the ladder/FBD networks
      _w1 : Bool;
   END_VAR
BEGIN

REGION Network 1: Sistema de Amostragem
   // O sistema irá realizar 4 amostra no periodo de 2s e realizar um filtro, contra interferências externas no sistema.
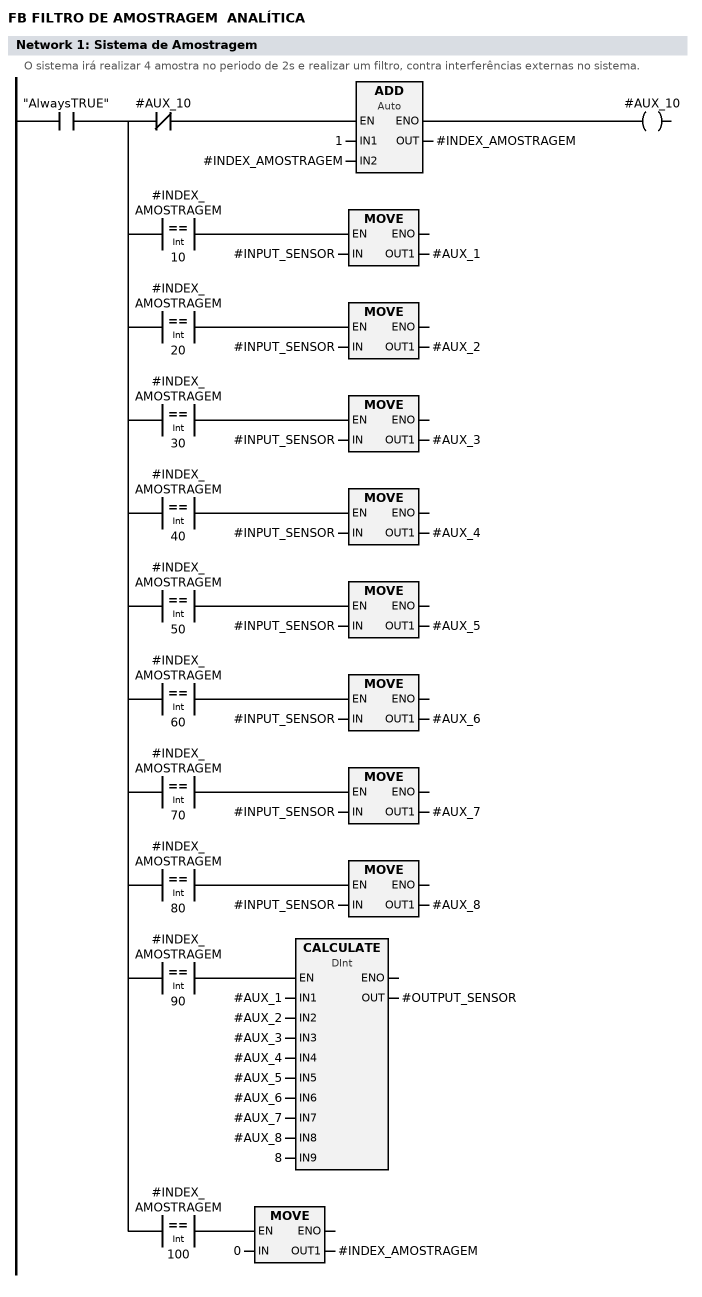
   RUNG wire#powerrail
      Contact( "AlwaysTRUE" )
      wire#w1
      I_Contact( #AUX_10 )
      Add(in1 := 1, in2 := #INDEX_AMOSTRAGEM, out => #INDEX_AMOSTRAGEM)
      Coil( #AUX_10 )
   END_RUNG
   RUNG wire#w1
      { S7_Templates := "SrcType := Int" } EQ_Contact(in1 := #INDEX_AMOSTRAGEM, in2 := 10)
      Move(in := #INPUT_SENSOR, out1 => #AUX_1)
   END_RUNG
   RUNG wire#w1
      { S7_Templates := "SrcType := Int" } EQ_Contact(in1 := #INDEX_AMOSTRAGEM, in2 := 20)
      Move(in := #INPUT_SENSOR, out1 => #AUX_2)
   END_RUNG
   RUNG wire#w1
      { S7_Templates := "SrcType := Int" } EQ_Contact(in1 := #INDEX_AMOSTRAGEM, in2 := 30)
      Move(in := #INPUT_SENSOR, out1 => #AUX_3)
   END_RUNG
   RUNG wire#w1
      { S7_Templates := "SrcType := Int" } EQ_Contact(in1 := #INDEX_AMOSTRAGEM, in2 := 40)
      Move(in := #INPUT_SENSOR, out1 => #AUX_4)
   END_RUNG
   RUNG wire#w1
      { S7_Templates := "SrcType := Int" } EQ_Contact(in1 := #INDEX_AMOSTRAGEM, in2 := 50)
      Move(in := #INPUT_SENSOR, out1 => #AUX_5)
   END_RUNG
   RUNG wire#w1
      { S7_Templates := "SrcType := Int" } EQ_Contact(in1 := #INDEX_AMOSTRAGEM, in2 := 60)
      Move(in := #INPUT_SENSOR, out1 => #AUX_6)
   END_RUNG
   RUNG wire#w1
      { S7_Templates := "SrcType := Int" } EQ_Contact(in1 := #INDEX_AMOSTRAGEM, in2 := 70)
      Move(in := #INPUT_SENSOR, out1 => #AUX_7)
   END_RUNG
   RUNG wire#w1
      { S7_Templates := "SrcType := Int" } EQ_Contact(in1 := #INDEX_AMOSTRAGEM, in2 := 80)
      Move(in := #INPUT_SENSOR, out1 => #AUX_8)
   END_RUNG
   RUNG wire#w1
      { S7_Templates := "SrcType := Int" } EQ_Contact(in1 := #INDEX_AMOSTRAGEM, in2 := 90)
      { S7_Templates := "SrcType := DInt"; S7_Expression := "(IN1+IN2+IN3+IN4+IN5+IN6+IN7+IN8)/IN9" } Calculate(in1 := #AUX_1, in2 := #AUX_2, in3 := #AUX_3, in4 := #AUX_4, in5 := #AUX_5, in6 := #AUX_6, in7 := #AUX_7, in8 := #AUX_8, in9 := 8, out => #OUTPUT_SENSOR)
   END_RUNG
   RUNG wire#w1
      { S7_Templates := "SrcType := Int" } EQ_Contact(in1 := #INDEX_AMOSTRAGEM, in2 := 100)
      Move(in := 0, out1 => #INDEX_AMOSTRAGEM)
   END_RUNG
   // the same network as SCL:
   #_w1 := "AlwaysTRUE" AND NOT #AUX_10;
   IF #_w1 THEN #INDEX_AMOSTRAGEM := 1 + #INDEX_AMOSTRAGEM; END_IF;
   #AUX_10 := #_w1;
   IF "AlwaysTRUE" AND (#INDEX_AMOSTRAGEM = 10) THEN #AUX_1 := #INPUT_SENSOR; END_IF;
   IF "AlwaysTRUE" AND (#INDEX_AMOSTRAGEM = 20) THEN #AUX_2 := #INPUT_SENSOR; END_IF;
   IF "AlwaysTRUE" AND (#INDEX_AMOSTRAGEM = 30) THEN #AUX_3 := #INPUT_SENSOR; END_IF;
   IF "AlwaysTRUE" AND (#INDEX_AMOSTRAGEM = 40) THEN #AUX_4 := #INPUT_SENSOR; END_IF;
   IF "AlwaysTRUE" AND (#INDEX_AMOSTRAGEM = 50) THEN #AUX_5 := #INPUT_SENSOR; END_IF;
   IF "AlwaysTRUE" AND (#INDEX_AMOSTRAGEM = 60) THEN #AUX_6 := #INPUT_SENSOR; END_IF;
   IF "AlwaysTRUE" AND (#INDEX_AMOSTRAGEM = 70) THEN #AUX_7 := #INPUT_SENSOR; END_IF;
   IF "AlwaysTRUE" AND (#INDEX_AMOSTRAGEM = 80) THEN #AUX_8 := #INPUT_SENSOR; END_IF;
   IF "AlwaysTRUE" AND (#INDEX_AMOSTRAGEM = 90) THEN
       #OUTPUT_SENSOR := (#AUX_1+#AUX_2+#AUX_3+#AUX_4+#AUX_5+#AUX_6+#AUX_7+#AUX_8)/8;
   END_IF;
   IF "AlwaysTRUE" AND (#INDEX_AMOSTRAGEM = 100) THEN #INDEX_AMOSTRAGEM := 0; END_IF;
END_REGION
END_FUNCTION_BLOCK

FUNCTION_BLOCK "FB LIMITES_OPERACAO_SENSOR"   // FB25, LAD
{ S7_Optimized_Access := 'TRUE' }
VERSION : 0.1
   VAR_INPUT
      STATUS_SENSOR : Real;
      COMANDO : Int;
      COMANDO_VALOR : Int;
      ENTRADA_VALOR_MUITO_BAIXO : Int;
      ENTRADA_VALOR_BAIXO : Int;
      ENTRADA_VALOR_ALTO : Int;
      ENTRADA_VALOR_MUITO_ALTO : Int;
      COMANDO_MANUTENCAO : Bool;
      SEM_SINAL_4mA : Bool;
   END_VAR
   VAR_OUTPUT
      SAIDA_LEITURA_MUITO_BAIXA : Bool;
      SAIDA_LEITURA_BAIXO : Bool;
      SAIDA_LEITURA_ALTO : Bool;
      SAIDA_LEITURA_MUITO_ALTO : Bool;
      VALOR_MUITO_BAIXO : Int;
      VALOR_BAIXO : Int;
      VALOR_ALTO : Int;
      VALOR_MUITO_ALTO : Int;
   END_VAR
   VAR
      TON_1 : IEC_TIMER;
      TON_2 : IEC_TIMER;
      TON_3 : IEC_TIMER;
      TON_4 : IEC_TIMER;
   END_VAR
   VAR_TEMP   // added for the SCL form of the ladder/FBD networks
      _w1 : Bool;
   END_VAR
BEGIN

REGION Network 1: Carrega valor de referencia
   // Network responsável por carregar os valores de referência (setpoints)
   //  para os limites do Medidor, com base em um comando de seleção de valor.
   //  O valor em '#COMANDO' determina qual conjunto de limites será ativo.
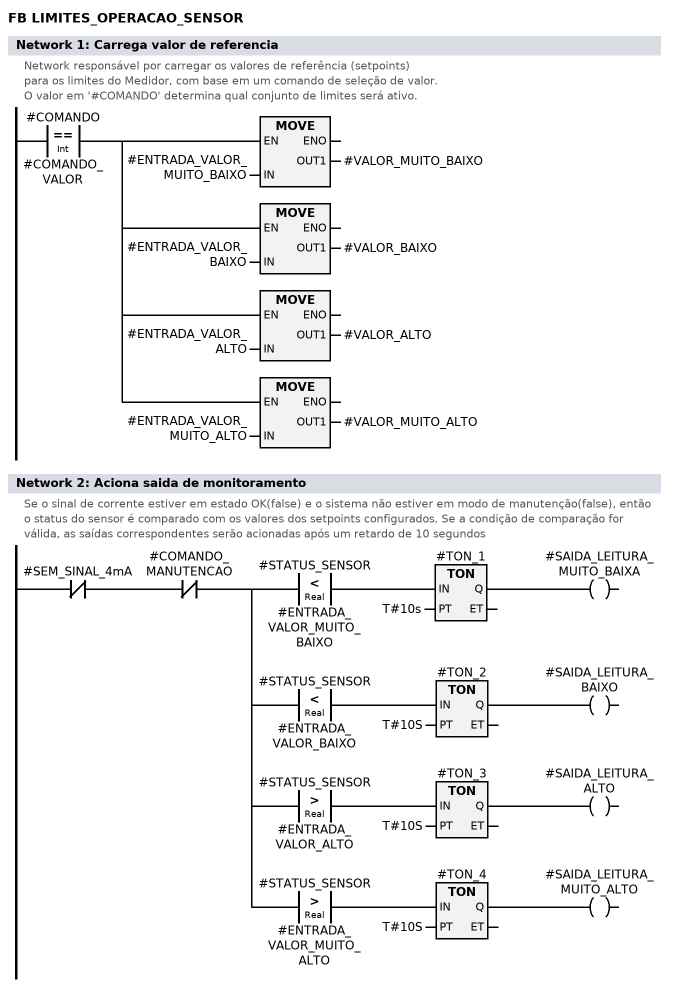
   RUNG wire#powerrail
      { S7_Templates := "SrcType := Int" } EQ_Contact(in1 := #COMANDO, in2 := #COMANDO_VALOR)
      wire#w1
      Move(in := #ENTRADA_VALOR_MUITO_BAIXO, out1 => #VALOR_MUITO_BAIXO)
   END_RUNG
   RUNG wire#w1
      Move(in := #ENTRADA_VALOR_BAIXO, out1 => #VALOR_BAIXO)
   END_RUNG
   RUNG wire#w1
      Move(in := #ENTRADA_VALOR_ALTO, out1 => #VALOR_ALTO)
   END_RUNG
   RUNG wire#w1
      Move(in := #ENTRADA_VALOR_MUITO_ALTO, out1 => #VALOR_MUITO_ALTO)
   END_RUNG
   // the same network as SCL:
   IF #COMANDO = #COMANDO_VALOR THEN
       #VALOR_MUITO_BAIXO := #ENTRADA_VALOR_MUITO_BAIXO;
       #VALOR_BAIXO := #ENTRADA_VALOR_BAIXO;
       #VALOR_ALTO := #ENTRADA_VALOR_ALTO;
       #VALOR_MUITO_ALTO := #ENTRADA_VALOR_MUITO_ALTO;
   END_IF;
END_REGION

REGION Network 2: Aciona saida de monitoramento
   // Se o sinal de corrente estiver em estado OK(false) e o sistema não estiver em modo de manutenção(false), então o status do sensor é comparado com os valores dos setpoints configurados. Se a condição de comparação for válida, as saídas correspondentes serão acionadas após um retardo de 10 segundos
   #_w1 := NOT #SEM_SINAL_4mA AND NOT #COMANDO_MANUTENCAO;
   #TON_1.TON(IN := #_w1 AND (#STATUS_SENSOR < #ENTRADA_VALOR_MUITO_BAIXO), PT := T#10s);
   #SAIDA_LEITURA_MUITO_BAIXA := #TON_1.Q;
   #TON_2.TON(IN := #_w1 AND (#STATUS_SENSOR < #ENTRADA_VALOR_BAIXO), PT := T#10S);
   #SAIDA_LEITURA_BAIXO := #TON_2.Q;
   #TON_3.TON(IN := #_w1 AND (#STATUS_SENSOR > #ENTRADA_VALOR_ALTO), PT := T#10S);
   #SAIDA_LEITURA_ALTO := #TON_3.Q;
   #TON_4.TON(IN := #_w1 AND (#STATUS_SENSOR > #ENTRADA_VALOR_MUITO_ALTO), PT := T#10S);
   #SAIDA_LEITURA_MUITO_ALTO := #TON_4.Q;
END_REGION
END_FUNCTION_BLOCK

FUNCTION_BLOCK "AUX_PID"   // FB31, LAD
{ S7_Optimized_Access := 'TRUE' }
VERSION : 0.1
// Esse bloco consiste em realizar um filtro para auxiliar na atuação do bloco PID
   VAR_INPUT
      SETPOINT_PID : Real;
      STATUS_VARIAVEL : Real;
      CADASTRO_LIMITE_MENOR : Real;
      CADASTRO_LIMITE_MAIOR : Real;
      CADASTRO_GANHO_PID_LIMITE : Real;
      CADASTRO_TEMPO_BLOCO_LIMITE : Real;
      CADASTRO_TEMPO_FORA_LIMITE : Real;
      CADASTRO_GANHO_FORA_LIMITE : Real;
   END_VAR
   VAR_OUTPUT
      GANHO_BLOCO : Real;
      TEMPO_BLOCO : Real;
   END_VAR
   VAR_TEMP
      LIMITE_MENOR : Real;
      LIMITE_MAIOR : Real;
   END_VAR
   VAR_TEMP   // added for the SCL form of the ladder/FBD networks
      _w1 : Bool;
   END_VAR
BEGIN

REGION Network 1
   // Se a variável de processo estiver dentro do limite, o bloco será configurado de forma lenta, reduzindo o overshoot.
   // Se a variável de processo estiver fora do limite, o bloco será configurado de forma rápida.
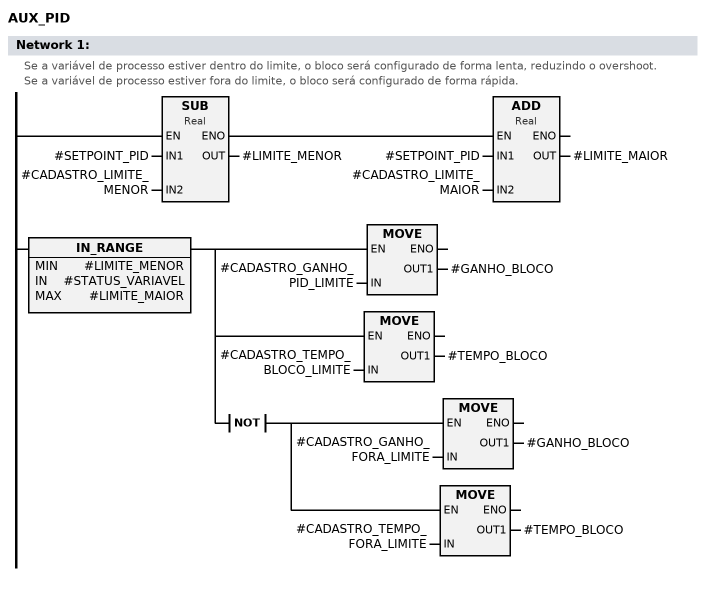
   RUNG wire#powerrail
      { S7_Templates := "SrcType := Real" } Sub(in1 := #SETPOINT_PID, in2 := #CADASTRO_LIMITE_MENOR, out => #LIMITE_MENOR)
      { S7_Templates := "SrcType := Real" } Add(in1 := #SETPOINT_PID, in2 := #CADASTRO_LIMITE_MAIOR, out => #LIMITE_MAIOR)
   END_RUNG
   RUNG wire#powerrail
      { S7_Templates := "SrcType := Real" } InRange(min := #LIMITE_MENOR, in := #STATUS_VARIAVEL, max := #LIMITE_MAIOR)
      wire#w1
      Move(in := #CADASTRO_GANHO_PID_LIMITE, out1 => #GANHO_BLOCO)
   END_RUNG
   RUNG wire#w1
      Move(in := #CADASTRO_TEMPO_BLOCO_LIMITE, out1 => #TEMPO_BLOCO)
   END_RUNG
   RUNG wire#w1
      Not()
      wire#w2
      Move(in := #CADASTRO_GANHO_FORA_LIMITE, out1 => #GANHO_BLOCO)
   END_RUNG
   RUNG wire#w2
      Move(in := #CADASTRO_TEMPO_FORA_LIMITE, out1 => #TEMPO_BLOCO)
   END_RUNG
   // the same network as SCL:
   #LIMITE_MENOR := #SETPOINT_PID - #CADASTRO_LIMITE_MENOR;
   #LIMITE_MAIOR := #SETPOINT_PID + #CADASTRO_LIMITE_MAIOR;
   #_w1 := (#LIMITE_MENOR <= #STATUS_VARIAVEL) AND (#STATUS_VARIAVEL <= #LIMITE_MAIOR);
   IF #_w1 THEN
       #GANHO_BLOCO := #CADASTRO_GANHO_PID_LIMITE;
       #TEMPO_BLOCO := #CADASTRO_TEMPO_BLOCO_LIMITE;
   END_IF;
   IF NOT #_w1 THEN
       #GANHO_BLOCO := #CADASTRO_GANHO_FORA_LIMITE;
       #TEMPO_BLOCO := #CADASTRO_TEMPO_FORA_LIMITE;
   END_IF;
END_REGION
END_FUNCTION_BLOCK

// folder: 1. FB Bilbiotecas/1.4 Alarmes e Falhas

FUNCTION_BLOCK "FB ALARME DIGITAL"   // FB3, LAD
TITLE = Function Block ALARME DIGITAL
{ S7_Optimized_Access := 'TRUE' }
VERSION : 0.1
// Tratamento de alarmes: Setando e Resetando sinais digitais relacionados aos alarmes
   VAR_INPUT
      Temp_Histerese : Time;
      SINAL_ENTRADA_DIGITAL_BIT_0 : Bool;   // Entrada digital do sinal elétrico
      SINAL_ENTRADA_DIGITAL_BIT_1 : Bool;
      SINAL_ENTRADA_DIGITAL_BIT_2 : Bool;
      SINAL_ENTRADA_DIGITAL_BIT_3 : Bool;
      SINAL_ENTRADA_DIGITAL_BIT_4 : Bool;
      SINAL_ENTRADA_DIGITAL_BIT_5 : Bool;
      SINAL_ENTRADA_DIGITAL_BIT_6 : Bool;
      SINAL_ENTRADA_DIGITAL_BIT_7 : Bool;
      SINAL_ENTRADA_DIGITAL_BIT_8 : Bool;
      SINAL_ENTRADA_DIGITAL_BIT_9 : Bool;
      SINAL_ENTRADA_DIGITAL_BIT_10 : Bool;
      SINAL_ENTRADA_DIGITAL_BIT_11 : Bool;
      SINAL_ENTRADA_DIGITAL_BIT_12 : Bool;
      SINAL_ENTRADA_DIGITAL_BIT_13 : Bool;
      SINAL_ENTRADA_DIGITAL_BIT_14 : Bool;
      SINAL_ENTRADA_DIGITAL_BIT_15 : Bool;
   END_VAR
   VAR_OUTPUT
      BD_GLOBAL_ALARME_BIT_0 : Bool;   // Saída digital instanciada no FB
      BD_GLOBAL_ALARME_BIT_1 : Bool;
      BD_GLOBAL_ALARME_BIT_2 : Bool;
      BD_GLOBAL_ALARME_BIT_3 : Bool;
      BD_GLOBAL_ALARME_BIT_4 : Bool;
      BD_GLOBAL_ALARME_BIT_5 : Bool;
      BD_GLOBAL_ALARME_BIT_6 : Bool;
      BD_GLOBAL_ALARME_BIT_7 : Bool;
      BD_GLOBAL_ALARME_BIT_8 : Bool;
      BD_GLOBAL_ALARME_BIT_9 : Bool;
      BD_GLOBAL_ALARME_BIT_10 : Bool;
      BD_GLOBAL_ALARME_BIT_11 : Bool;
      BD_GLOBAL_ALARME_BIT_12 : Bool;
      BD_GLOBAL_ALARME_BIT_13 : Bool;
      BD_GLOBAL_ALARME_BIT_14 : Bool;
      BD_GLOBAL_ALARME_BIT_15 : Bool;
   END_VAR
   VAR
      RESET_TIME_0 : IEC_TIMER;   // Reset do alarme caso o sinal seja interrompido
      RESET_TIME_1 : TON_TIME;
      RESET_TIME_2 : TON_TIME;
      RESET_TIME_3 : TON_TIME;
      RESET_TIME_4 : TON_TIME;
      RESET_TIME_5 : TON_TIME;
      RESET_TIME_6 : TON_TIME;
      RESET_TIME_7 : TON_TIME;
      RESET_TIME_8 : TON_TIME;
      RESET_TIME_9 : TON_TIME;
      RESET_TIME_10 : TON_TIME;
      RESET_TIME_11 : TON_TIME;
      RESET_TIME_12 : TON_TIME;
      RESET_TIME_13 : TON_TIME;
      RESET_TIME_14 : TON_TIME;
      RESET_TIME_15 : TON_TIME;
      ACIONA_BD_ALARME_0 : Bool;   // Chaveamento para acionar/desacionar o alarme
      ACIONA_BD_ALARME_1 : Bool;
      ACIONA_BD_ALARME_2 : Bool;
      ACIONA_BD_ALARME_3 : Bool;
      ACIONA_BD_ALARME_4 : Bool;
      ACIONA_BD_ALARME_5 : Bool;
      ACIONA_BD_ALARME_6 : Bool;
      ACIONA_BD_ALARME_7 : Bool;
      ACIONA_BD_ALARME_8 : Bool;
      ACIONA_BD_ALARME_9 : Bool;
      ACIONA_BD_ALARME_10 : Bool;
      ACIONA_BD_ALARME_11 : Bool;
      ACIONA_BD_ALARME_12 : Bool;
      ACIONA_BD_ALARME_13 : Bool;
      ACIONA_BD_ALARME_14 : Bool;
      ACIONA_BD_ALARME_15 : Bool;
   END_VAR
BEGIN

REGION Network 1: SET RESET
   // Recebendo sinal da I/O do equipamento e setando o alarme dentro da DB. Após a entrada identificar nível baixo (0) a saída do alarme é resetada conforme tempo configurado.
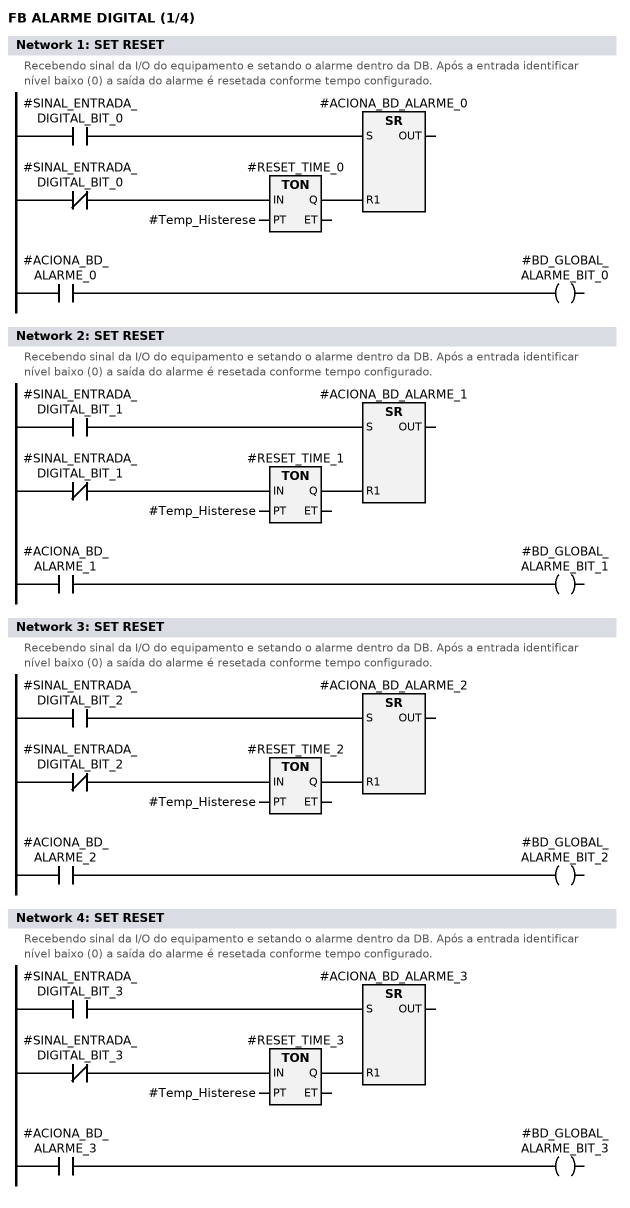
   #RESET_TIME_0.TON(IN := NOT #SINAL_ENTRADA_DIGITAL_BIT_0, PT := #Temp_Histerese);
   IF #SINAL_ENTRADA_DIGITAL_BIT_0 THEN
       #ACIONA_BD_ALARME_0 := TRUE;   // SR flip-flop
   END_IF;
   IF #RESET_TIME_0.Q THEN #ACIONA_BD_ALARME_0 := FALSE; END_IF;
   #BD_GLOBAL_ALARME_BIT_0 := #ACIONA_BD_ALARME_0;
END_REGION

REGION Network 2: SET RESET
   // Recebendo sinal da I/O do equipamento e setando o alarme dentro da DB. Após a entrada identificar nível baixo (0) a saída do alarme é resetada conforme tempo configurado.
   #RESET_TIME_1(IN := NOT #SINAL_ENTRADA_DIGITAL_BIT_1, PT := #Temp_Histerese);   // TON
   IF #SINAL_ENTRADA_DIGITAL_BIT_1 THEN
       #ACIONA_BD_ALARME_1 := TRUE;   // SR flip-flop
   END_IF;
   IF #RESET_TIME_1.Q THEN #ACIONA_BD_ALARME_1 := FALSE; END_IF;
   #BD_GLOBAL_ALARME_BIT_1 := #ACIONA_BD_ALARME_1;
END_REGION

REGION Network 3: SET RESET
   // Recebendo sinal da I/O do equipamento e setando o alarme dentro da DB. Após a entrada identificar nível baixo (0) a saída do alarme é resetada conforme tempo configurado.
   #RESET_TIME_2(IN := NOT #SINAL_ENTRADA_DIGITAL_BIT_2, PT := #Temp_Histerese);   // TON
   IF #SINAL_ENTRADA_DIGITAL_BIT_2 THEN
       #ACIONA_BD_ALARME_2 := TRUE;   // SR flip-flop
   END_IF;
   IF #RESET_TIME_2.Q THEN #ACIONA_BD_ALARME_2 := FALSE; END_IF;
   #BD_GLOBAL_ALARME_BIT_2 := #ACIONA_BD_ALARME_2;
END_REGION

REGION Network 4: SET RESET
   // Recebendo sinal da I/O do equipamento e setando o alarme dentro da DB. Após a entrada identificar nível baixo (0) a saída do alarme é resetada conforme tempo configurado.
   #RESET_TIME_3(IN := NOT #SINAL_ENTRADA_DIGITAL_BIT_3, PT := #Temp_Histerese);   // TON
   IF #SINAL_ENTRADA_DIGITAL_BIT_3 THEN
       #ACIONA_BD_ALARME_3 := TRUE;   // SR flip-flop
   END_IF;
   IF #RESET_TIME_3.Q THEN #ACIONA_BD_ALARME_3 := FALSE; END_IF;
   #BD_GLOBAL_ALARME_BIT_3 := #ACIONA_BD_ALARME_3;
END_REGION

REGION Network 5: SET RESET
   // Recebendo sinal da I/O do equipamento e setando o alarme dentro da DB. Após a entrada identificar nível baixo (0) a saída do alarme é resetada conforme tempo configurado.
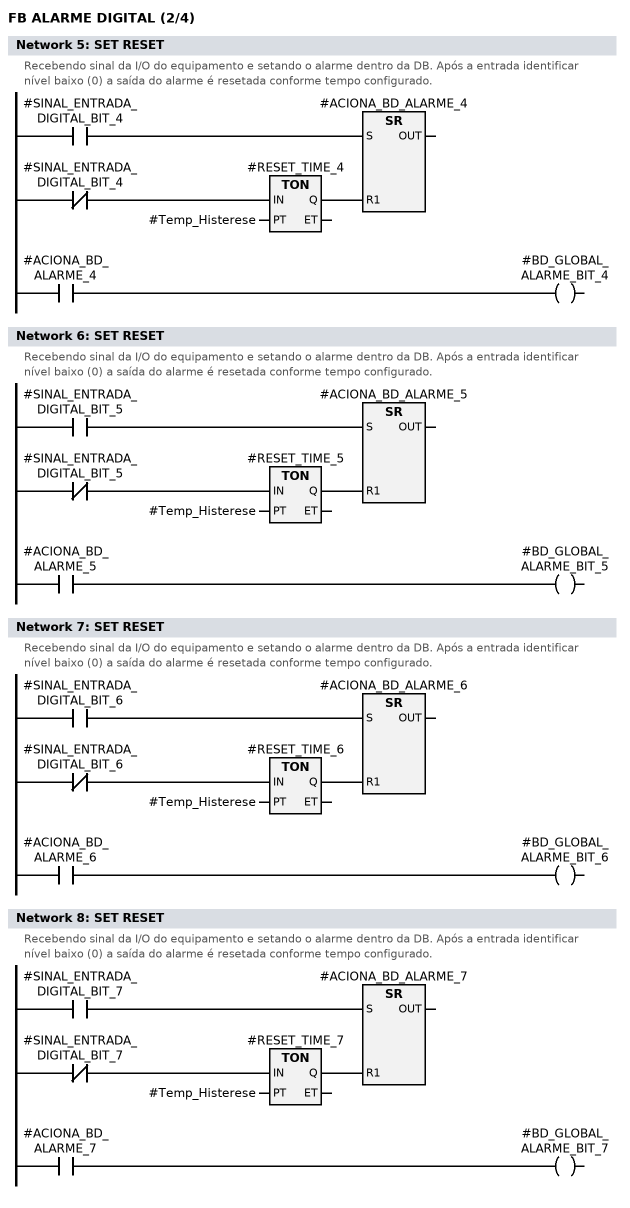
   #RESET_TIME_4(IN := NOT #SINAL_ENTRADA_DIGITAL_BIT_4, PT := #Temp_Histerese);   // TON
   IF #SINAL_ENTRADA_DIGITAL_BIT_4 THEN
       #ACIONA_BD_ALARME_4 := TRUE;   // SR flip-flop
   END_IF;
   IF #RESET_TIME_4.Q THEN #ACIONA_BD_ALARME_4 := FALSE; END_IF;
   #BD_GLOBAL_ALARME_BIT_4 := #ACIONA_BD_ALARME_4;
END_REGION

REGION Network 6: SET RESET
   // Recebendo sinal da I/O do equipamento e setando o alarme dentro da DB. Após a entrada identificar nível baixo (0) a saída do alarme é resetada conforme tempo configurado.
   #RESET_TIME_5(IN := NOT #SINAL_ENTRADA_DIGITAL_BIT_5, PT := #Temp_Histerese);   // TON
   IF #SINAL_ENTRADA_DIGITAL_BIT_5 THEN
       #ACIONA_BD_ALARME_5 := TRUE;   // SR flip-flop
   END_IF;
   IF #RESET_TIME_5.Q THEN #ACIONA_BD_ALARME_5 := FALSE; END_IF;
   #BD_GLOBAL_ALARME_BIT_5 := #ACIONA_BD_ALARME_5;
END_REGION

REGION Network 7: SET RESET
   // Recebendo sinal da I/O do equipamento e setando o alarme dentro da DB. Após a entrada identificar nível baixo (0) a saída do alarme é resetada conforme tempo configurado.
   #RESET_TIME_6(IN := NOT #SINAL_ENTRADA_DIGITAL_BIT_6, PT := #Temp_Histerese);   // TON
   IF #SINAL_ENTRADA_DIGITAL_BIT_6 THEN
       #ACIONA_BD_ALARME_6 := TRUE;   // SR flip-flop
   END_IF;
   IF #RESET_TIME_6.Q THEN #ACIONA_BD_ALARME_6 := FALSE; END_IF;
   #BD_GLOBAL_ALARME_BIT_6 := #ACIONA_BD_ALARME_6;
END_REGION

REGION Network 8: SET RESET
   // Recebendo sinal da I/O do equipamento e setando o alarme dentro da DB. Após a entrada identificar nível baixo (0) a saída do alarme é resetada conforme tempo configurado.
   #RESET_TIME_7(IN := NOT #SINAL_ENTRADA_DIGITAL_BIT_7, PT := #Temp_Histerese);   // TON
   IF #SINAL_ENTRADA_DIGITAL_BIT_7 THEN
       #ACIONA_BD_ALARME_7 := TRUE;   // SR flip-flop
   END_IF;
   IF #RESET_TIME_7.Q THEN #ACIONA_BD_ALARME_7 := FALSE; END_IF;
   #BD_GLOBAL_ALARME_BIT_7 := #ACIONA_BD_ALARME_7;
END_REGION

REGION Network 9: SET RESET
   // Recebendo sinal da I/O do equipamento e setando o alarme dentro da DB. Após a entrada identificar nível baixo (0) a saída do alarme é resetada conforme tempo configurado.
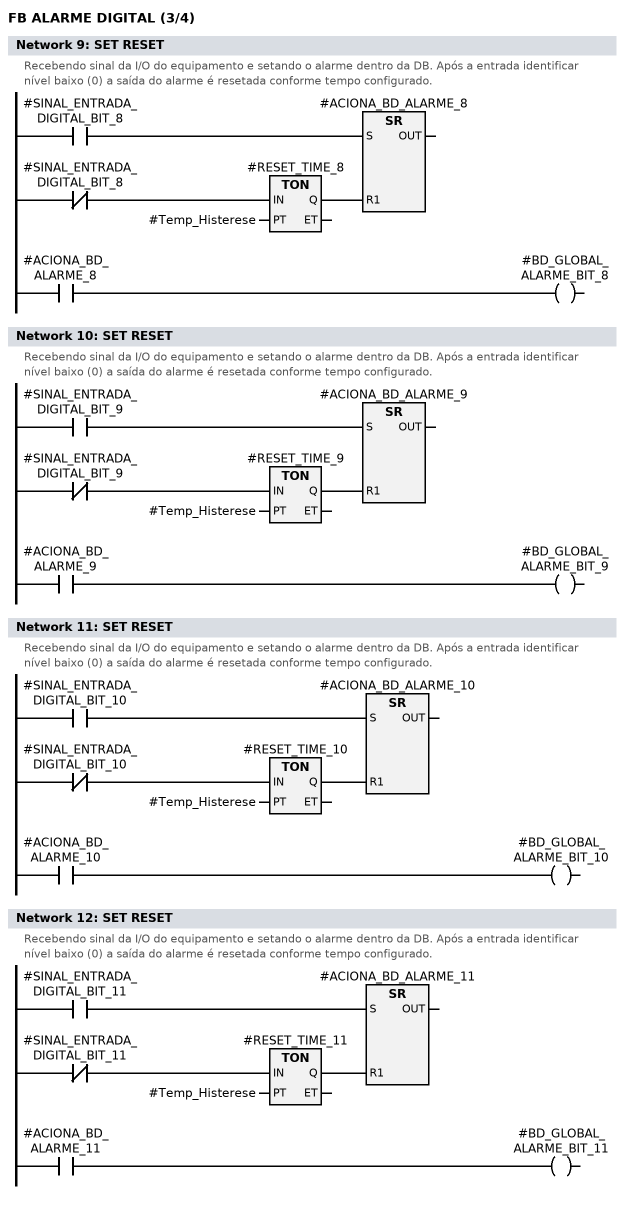
   #RESET_TIME_8(IN := NOT #SINAL_ENTRADA_DIGITAL_BIT_8, PT := #Temp_Histerese);   // TON
   IF #SINAL_ENTRADA_DIGITAL_BIT_8 THEN
       #ACIONA_BD_ALARME_8 := TRUE;   // SR flip-flop
   END_IF;
   IF #RESET_TIME_8.Q THEN #ACIONA_BD_ALARME_8 := FALSE; END_IF;
   #BD_GLOBAL_ALARME_BIT_8 := #ACIONA_BD_ALARME_8;
END_REGION

REGION Network 10: SET RESET
   // Recebendo sinal da I/O do equipamento e setando o alarme dentro da DB. Após a entrada identificar nível baixo (0) a saída do alarme é resetada conforme tempo configurado.
   #RESET_TIME_9(IN := NOT #SINAL_ENTRADA_DIGITAL_BIT_9, PT := #Temp_Histerese);   // TON
   IF #SINAL_ENTRADA_DIGITAL_BIT_9 THEN
       #ACIONA_BD_ALARME_9 := TRUE;   // SR flip-flop
   END_IF;
   IF #RESET_TIME_9.Q THEN #ACIONA_BD_ALARME_9 := FALSE; END_IF;
   #BD_GLOBAL_ALARME_BIT_9 := #ACIONA_BD_ALARME_9;
END_REGION

REGION Network 11: SET RESET
   // Recebendo sinal da I/O do equipamento e setando o alarme dentro da DB. Após a entrada identificar nível baixo (0) a saída do alarme é resetada conforme tempo configurado.
   #RESET_TIME_10(IN := NOT #SINAL_ENTRADA_DIGITAL_BIT_10, PT := #Temp_Histerese);   // TON
   IF #SINAL_ENTRADA_DIGITAL_BIT_10 THEN
       #ACIONA_BD_ALARME_10 := TRUE;   // SR flip-flop
   END_IF;
   IF #RESET_TIME_10.Q THEN #ACIONA_BD_ALARME_10 := FALSE; END_IF;
   #BD_GLOBAL_ALARME_BIT_10 := #ACIONA_BD_ALARME_10;
END_REGION

REGION Network 12: SET RESET
   // Recebendo sinal da I/O do equipamento e setando o alarme dentro da DB. Após a entrada identificar nível baixo (0) a saída do alarme é resetada conforme tempo configurado.
   #RESET_TIME_11(IN := NOT #SINAL_ENTRADA_DIGITAL_BIT_11, PT := #Temp_Histerese);   // TON
   IF #SINAL_ENTRADA_DIGITAL_BIT_11 THEN
       #ACIONA_BD_ALARME_11 := TRUE;   // SR flip-flop
   END_IF;
   IF #RESET_TIME_11.Q THEN #ACIONA_BD_ALARME_11 := FALSE; END_IF;
   #BD_GLOBAL_ALARME_BIT_11 := #ACIONA_BD_ALARME_11;
END_REGION

REGION Network 13: SET RESET
   // Recebendo sinal da I/O do equipamento e setando o alarme dentro da DB. Após a entrada identificar nível baixo (0) a saída do alarme é resetada conforme tempo configurado.
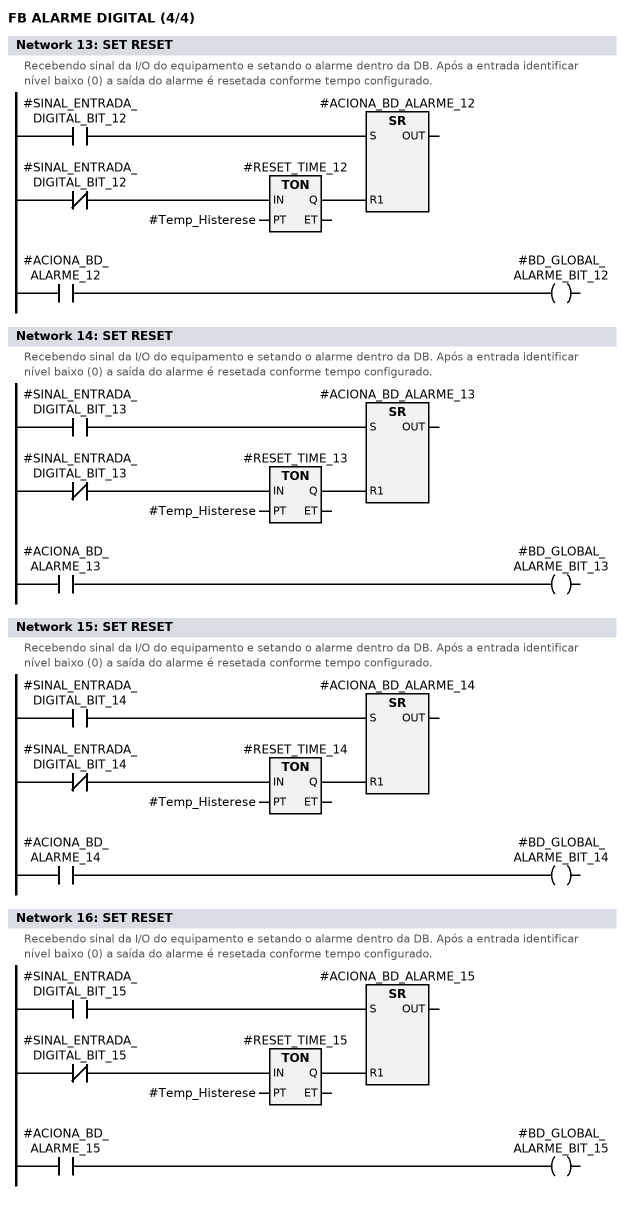
   #RESET_TIME_12(IN := NOT #SINAL_ENTRADA_DIGITAL_BIT_12, PT := #Temp_Histerese);   // TON
   IF #SINAL_ENTRADA_DIGITAL_BIT_12 THEN
       #ACIONA_BD_ALARME_12 := TRUE;   // SR flip-flop
   END_IF;
   IF #RESET_TIME_12.Q THEN #ACIONA_BD_ALARME_12 := FALSE; END_IF;
   #BD_GLOBAL_ALARME_BIT_12 := #ACIONA_BD_ALARME_12;
END_REGION

REGION Network 14: SET RESET
   // Recebendo sinal da I/O do equipamento e setando o alarme dentro da DB. Após a entrada identificar nível baixo (0) a saída do alarme é resetada conforme tempo configurado.
   #RESET_TIME_13(IN := NOT #SINAL_ENTRADA_DIGITAL_BIT_13, PT := #Temp_Histerese);   // TON
   IF #SINAL_ENTRADA_DIGITAL_BIT_13 THEN
       #ACIONA_BD_ALARME_13 := TRUE;   // SR flip-flop
   END_IF;
   IF #RESET_TIME_13.Q THEN #ACIONA_BD_ALARME_13 := FALSE; END_IF;
   #BD_GLOBAL_ALARME_BIT_13 := #ACIONA_BD_ALARME_13;
END_REGION

REGION Network 15: SET RESET
   // Recebendo sinal da I/O do equipamento e setando o alarme dentro da DB. Após a entrada identificar nível baixo (0) a saída do alarme é resetada conforme tempo configurado.
   #RESET_TIME_14(IN := NOT #SINAL_ENTRADA_DIGITAL_BIT_14, PT := #Temp_Histerese);   // TON
   IF #SINAL_ENTRADA_DIGITAL_BIT_14 THEN
       #ACIONA_BD_ALARME_14 := TRUE;   // SR flip-flop
   END_IF;
   IF #RESET_TIME_14.Q THEN #ACIONA_BD_ALARME_14 := FALSE; END_IF;
   #BD_GLOBAL_ALARME_BIT_14 := #ACIONA_BD_ALARME_14;
END_REGION

REGION Network 16: SET RESET
   // Recebendo sinal da I/O do equipamento e setando o alarme dentro da DB. Após a entrada identificar nível baixo (0) a saída do alarme é resetada conforme tempo configurado.
   #RESET_TIME_15(IN := NOT #SINAL_ENTRADA_DIGITAL_BIT_15, PT := #Temp_Histerese);   // TON
   IF #SINAL_ENTRADA_DIGITAL_BIT_15 THEN
       #ACIONA_BD_ALARME_15 := TRUE;   // SR flip-flop
   END_IF;
   IF #RESET_TIME_15.Q THEN #ACIONA_BD_ALARME_15 := FALSE; END_IF;
   #BD_GLOBAL_ALARME_BIT_15 := #ACIONA_BD_ALARME_15;
END_REGION
END_FUNCTION_BLOCK

FUNCTION_BLOCK "FB FALHA"   // FB9, LAD
TITLE = Function Block FALHA - Falha dos motores/bombas
{ S7_Optimized_Access := 'TRUE' }
VERSION : 0.1
// Network 1: Condição SET-RESET da Falha da bomba
   VAR_INPUT
      INPUT_FALHA : Bool;   // Entrada do sinal de falha instanciado na Network 1
      INPUT_FILTRO_PARA_FALHA : Time;
      INPUT_TEMPO_RESET : Time;   // Tempo em segundos que a bomba irá resetar após identificar sem falha
      INPUT_TEMPO_NÃO_LIGOU : Time;   // Se após ligar a bomba não retornar o sinal de LIGADO pelo tempo configurado, aciona falha
      INPUT_LIGADO : Bool;   // Entrada do sinal de Motor/Bomba ligado
      INPUT_RESET_FALHA : Bool;   // Resetar a falha manualmente caso o sinal de INPUT_FALHA esteja FALSE
      INPUT_REMOTO_AUTO : Bool;
      INPUT_TEMPO_RESET_AUTO : Time;
      INPUT_SAIDA_LIGA_BOMBA : Bool;   // Saída para ligar a bomba acionada
      INPUT_HABILITA_CONJUNTO : Bool;   // Identificação do conjunto de bombas (principal e reserva)
      INPUT_MANUTENCAO : Bool;   // Entrada responsavel por mudar o estado do equipamento em manut, sendo sem falha ativa.
   END_VAR
   VAR_OUTPUT
      FALHA : Bool;   // Saída do sinal de falha da instância do FB para o FC
      RESET_FALHA_INVERSOR : Bool;   // Reset sinal de falha do inversor de frequência
      FALHA_NÃO_LIGOU : Bool;
   END_VAR
   VAR
      NÃO_LIGOU : Bool;   // Sinal indicando que a bomba não ligou após comando, entrando em falha
      SET_FALHA : Bool;   // Memória auxiliar para o recebimento da falha
      TIMER_0 : IEC_TIMER;
      TIMER_1 : IEC_TIMER;   // Temporizador para resetar a Falha
      TIMER_2 : IEC_TIMER;   // Temporizador para entrar em Falha
      TIMER_3 : IEC_TIMER;   // Temporizador para entrar em Falha
      LIGA_BOMBA_AUX : Bool;   // Memória auxiliar para disparo do final de falha
   END_VAR
   VAR_TEMP   // added for the SCL form of the ladder/FBD networks
      _w1 : Bool;
   END_VAR
BEGIN

REGION Network 1: Saída do sinal de falha da instância do FB para o FC
   // Tratamento de falha da bomba
   // INPUT_FALHA: Entrada do sinal de falha instanciado na Network 1.
   // INPUT_TEMPO_RESET: Tempo em segundos que a bomba irá resetar após identificar sem falha.
   // INPUT_TEMPO_NÃO_LIGOU: Se após ligar a bomba não retornar o sinal de LIGADO pelo tempo configurado, aciona falha.
   // INPUT_LIGADO: Entrada do sinal de Motor/Bomba ligado
   // INPUT_RESET_FALHA: Resetar a falha manualmente caso o sinal de INPUT_FALHA esteja FALSE
   // NÃO_LIGOU: Memória auxiliar para acionar falha caso a bomba não retorno seu status de ligada.
